DATA_BLOCK "DB92_OP_Data"
{ S7_Optimized_Access := 'FALSE' }
VERSION : 0.1
NON_RETAIN
   STRUCT
      LocTime {InstructionName := 'DTL'; LibVersion := '1.0'} : DTL;
      tm_Array : Array[0..11] of Byte;
      Msg_B0 : Array[0..63] of Word;
      CtrlJob : Array[0..3] of Word;   // Steuerungsauftragsfach
      PicNum : Array[0..4] of Word;   // Steuerungsauftragsfach
      SPS_Idx : Int;   // Index eigene SPS
      Antr_Idx : Int;   // Index ausgewählter Antrieb für Anzeige/Bedienung
      Antr_Typ : Int;   // Typ ausgewählter Antrieb für Anzeige/Bedienung
      UserPrio : Int;   // Prio 0 - keine Bedienung, Prio 1 - Antrieb einzel, Prio 2 - alle Antriebe auf Bed. UV, Prio 3 - Parametrierung
      Antr_loc_prev : Bool;   // vorhergehenden (lokal) Antrieb in Panel-Auswahl anzeigen
      Antr_loc_next : Bool;   // nächsten Antrieb (lokal) in Panel-Auswahl anzeigen
      Antr_rem_prev : Bool;   // vorhergehenden (fern) Antrieb in Panel-Auswahl anzeigen
      Antr_rem_next : Bool;   // nächsten Antrieb (fern) in Panel-Auswahl anzeigen
      UserChg : Bool;   // Panelbenutzer hat gewechselt -> remote login prüfen
      PicSet_Antr_Menu : Bool;   // UV spezifisches Menü Antriebe aufrufen
      PicSet_Antr_Prm : Bool;   // Parameterbild zum gewählten Antrieb aufrufen
      MsgQuit : Bool;   // Quittierung Meldesystem
      Antr_Text_Idx_vis : Int;   // Textlisten für Bezeichnungen - Index für Auswahl Subliste 0..3
      Antr_Text_Idx_W0 : DWord;   // Textlisten für Bezeichnungen - Subliste 0
      Antr_Text_Idx_W1 : DWord;   // Textlisten für Bezeichnungen - Subliste 1
      Antr_Text_Idx_W2 : DWord;   // Textlisten für Bezeichnungen - Subliste 2
      Antr_Text_Idx_W3 : DWord;   // Textlisten für Bezeichnungen - Subliste 3
      UserID_BitIdx : DWord;   // Benutzerkennung bitweise, ID1=Bit 1 usw.
      Antr_UV_Idx : Byte;   // Index UV des gewählten Antriebs -> Anzeige, wenn nicht in eigener SPS abgearbeitet
      SPS_Idx_BitIdx : Byte;   // Index eigene SPS - Bitliste
      Antr_UV_rem : Bool;   // Hinweisfeld, wenn Antrieb in remoter SPS bearbeitet wird
      Antr_Bed_Sperr_0 : Array[0..63] of Bool;
      Antr_Bed_Sperr_1 : Array[0..63] of Bool;
      Bed_NHV : Array[1..128] of Bool;   // Bedienberechtigungen für (ferne) OP Bedienung
      activeUserGroup : Int;
   END_STRUCT;


BEGIN

END_DATA_BLOCK

DATA_BLOCK "DB93_AntrIdx"
{ S7_Optimized_Access := 'FALSE' }
VERSION : 0.1
NON_RETAIN
   STRUCT
      MaxIdx_ges : Int;
      MaxIdx : Array[0..6] of Byte;
      UV2ZEN : Array[0..6, 1..32] of Byte;
      ZEN2UV : Array[0..6, 1..132] of Byte;
      ANTR2UV : Array[1..132] of Byte;
      ANTR2OP : Array[1..132] of Byte;
      ANTR2TYP : Array[1..132] of Byte;
   END_STRUCT;


BEGIN
   MaxIdx_ges := 22;
   MaxIdx[0] := 16#00;
   MaxIdx[1] := 16#00;
   MaxIdx[2] := 16#16;
   MaxIdx[3] := 16#00;
   MaxIdx[4] := 16#00;
   MaxIdx[5] := 16#00;
   MaxIdx[6] := 16#00;
   UV2ZEN[0,1] := 16#00;
   UV2ZEN[0,2] := 16#00;
   UV2ZEN[0,3] := 16#00;
   UV2ZEN[0,4] := 16#00;
   UV2ZEN[0,5] := 16#00;
   UV2ZEN[0,6] := 16#00;
   UV2ZEN[0,7] := 16#00;
   UV2ZEN[0,8] := 16#00;
   UV2ZEN[0,9] := 16#00;
   UV2ZEN[0,10] := 16#00;
   UV2ZEN[0,11] := 16#00;
   UV2ZEN[0,12] := 16#00;
   UV2ZEN[0,13] := 16#00;
   UV2ZEN[0,14] := 16#00;
   UV2ZEN[0,15] := 16#00;
   UV2ZEN[0,16] := 16#00;
   UV2ZEN[0,17] := 16#00;
   UV2ZEN[0,18] := 16#00;
   UV2ZEN[0,19] := 16#00;
   UV2ZEN[0,20] := 16#00;
   UV2ZEN[0,21] := 16#00;
   UV2ZEN[0,22] := 16#00;
   UV2ZEN[0,23] := 16#00;
   UV2ZEN[0,24] := 16#00;
   UV2ZEN[0,25] := 16#00;
   UV2ZEN[0,26] := 16#00;
   UV2ZEN[0,27] := 16#00;
   UV2ZEN[0,28] := 16#00;
   UV2ZEN[0,29] := 16#00;
   UV2ZEN[0,30] := 16#00;
   UV2ZEN[0,31] := 16#00;
   UV2ZEN[0,32] := 16#00;
   UV2ZEN[1,1] := 16#00;
   UV2ZEN[1,2] := 16#00;
   UV2ZEN[1,3] := 16#00;
   UV2ZEN[1,4] := 16#00;
   UV2ZEN[1,5] := 16#00;
   UV2ZEN[1,6] := 16#00;
   UV2ZEN[1,7] := 16#00;
   UV2ZEN[1,8] := 16#00;
   UV2ZEN[1,9] := 16#00;
   UV2ZEN[1,10] := 16#00;
   UV2ZEN[1,11] := 16#00;
   UV2ZEN[1,12] := 16#00;
   UV2ZEN[1,13] := 16#00;
   UV2ZEN[1,14] := 16#00;
   UV2ZEN[1,15] := 16#00;
   UV2ZEN[1,16] := 16#00;
   UV2ZEN[1,17] := 16#00;
   UV2ZEN[1,18] := 16#00;
   UV2ZEN[1,19] := 16#00;
   UV2ZEN[1,20] := 16#00;
   UV2ZEN[1,21] := 16#00;
   UV2ZEN[1,22] := 16#00;
   UV2ZEN[1,23] := 16#00;
   UV2ZEN[1,24] := 16#00;
   UV2ZEN[1,25] := 16#00;
   UV2ZEN[1,26] := 16#00;
   UV2ZEN[1,27] := 16#00;
   UV2ZEN[1,28] := 16#00;
   UV2ZEN[1,29] := 16#00;
   UV2ZEN[1,30] := 16#00;
   UV2ZEN[1,31] := 16#00;
   UV2ZEN[1,32] := 16#00;
   UV2ZEN[2,1] := 16#01;
   UV2ZEN[2,2] := 16#02;
   UV2ZEN[2,3] := 16#03;
   UV2ZEN[2,4] := 16#04;
   UV2ZEN[2,5] := 16#05;
   UV2ZEN[2,6] := 16#06;
   UV2ZEN[2,7] := 16#07;
   UV2ZEN[2,8] := 16#08;
   UV2ZEN[2,9] := 16#09;
   UV2ZEN[2,10] := 16#0A;
   UV2ZEN[2,11] := 16#0B;
   UV2ZEN[2,12] := 16#0C;
   UV2ZEN[2,13] := 16#0D;
   UV2ZEN[2,14] := 16#0E;
   UV2ZEN[2,15] := 16#0F;
   UV2ZEN[2,16] := 16#10;
   UV2ZEN[2,17] := 16#11;
   UV2ZEN[2,18] := 16#12;
   UV2ZEN[2,19] := 16#13;
   UV2ZEN[2,20] := 16#14;
   UV2ZEN[2,21] := 16#15;
   UV2ZEN[2,22] := 16#16;
   UV2ZEN[2,23] := 16#00;
   UV2ZEN[2,24] := 16#00;
   UV2ZEN[2,25] := 16#00;
   UV2ZEN[2,26] := 16#00;
   UV2ZEN[2,27] := 16#00;
   UV2ZEN[2,28] := 16#00;
   UV2ZEN[2,29] := 16#00;
   UV2ZEN[2,30] := 16#00;
   UV2ZEN[2,31] := 16#00;
   UV2ZEN[2,32] := 16#00;
   UV2ZEN[3,1] := 16#00;
   UV2ZEN[3,2] := 16#00;
   UV2ZEN[3,3] := 16#00;
   UV2ZEN[3,4] := 16#00;
   UV2ZEN[3,5] := 16#00;
   UV2ZEN[3,6] := 16#00;
   UV2ZEN[3,7] := 16#00;
   UV2ZEN[3,8] := 16#00;
   UV2ZEN[3,9] := 16#00;
   UV2ZEN[3,10] := 16#00;
   UV2ZEN[3,11] := 16#00;
   UV2ZEN[3,12] := 16#00;
   UV2ZEN[3,13] := 16#00;
   UV2ZEN[3,14] := 16#00;
   UV2ZEN[3,15] := 16#00;
   UV2ZEN[3,16] := 16#00;
   UV2ZEN[3,17] := 16#00;
   UV2ZEN[3,18] := 16#00;
   UV2ZEN[3,19] := 16#00;
   UV2ZEN[3,20] := 16#00;
   UV2ZEN[3,21] := 16#00;
   UV2ZEN[3,22] := 16#00;
   UV2ZEN[3,23] := 16#00;
   UV2ZEN[3,24] := 16#00;
   UV2ZEN[3,25] := 16#00;
   UV2ZEN[3,26] := 16#00;
   UV2ZEN[3,27] := 16#00;
   UV2ZEN[3,28] := 16#00;
   UV2ZEN[3,29] := 16#00;
   UV2ZEN[3,30] := 16#00;
   UV2ZEN[3,31] := 16#00;
   UV2ZEN[3,32] := 16#00;
   UV2ZEN[4,1] := 16#00;
   UV2ZEN[4,2] := 16#00;
   UV2ZEN[4,3] := 16#00;
   UV2ZEN[4,4] := 16#00;
   UV2ZEN[4,5] := 16#00;
   UV2ZEN[4,6] := 16#00;
   UV2ZEN[4,7] := 16#00;
   UV2ZEN[4,8] := 16#00;
   UV2ZEN[4,9] := 16#00;
   UV2ZEN[4,10] := 16#00;
   UV2ZEN[4,11] := 16#00;
   UV2ZEN[4,12] := 16#00;
   UV2ZEN[4,13] := 16#00;
   UV2ZEN[4,14] := 16#00;
   UV2ZEN[4,15] := 16#00;
   UV2ZEN[4,16] := 16#00;
   UV2ZEN[4,17] := 16#00;
   UV2ZEN[4,18] := 16#00;
   UV2ZEN[4,19] := 16#00;
   UV2ZEN[4,20] := 16#00;
   UV2ZEN[4,21] := 16#00;
   UV2ZEN[4,22] := 16#00;
   UV2ZEN[4,23] := 16#00;
   UV2ZEN[4,24] := 16#00;
   UV2ZEN[4,25] := 16#00;
   UV2ZEN[4,26] := 16#00;
   UV2ZEN[4,27] := 16#00;
   UV2ZEN[4,28] := 16#00;
   UV2ZEN[4,29] := 16#00;
   UV2ZEN[4,30] := 16#00;
   UV2ZEN[4,31] := 16#00;
   UV2ZEN[4,32] := 16#00;
   UV2ZEN[5,1] := 16#00;
   UV2ZEN[5,2] := 16#00;
   UV2ZEN[5,3] := 16#00;
   UV2ZEN[5,4] := 16#00;
   UV2ZEN[5,5] := 16#00;
   UV2ZEN[5,6] := 16#00;
   UV2ZEN[5,7] := 16#00;
   UV2ZEN[5,8] := 16#00;
   UV2ZEN[5,9] := 16#00;
   UV2ZEN[5,10] := 16#00;
   UV2ZEN[5,11] := 16#00;
   UV2ZEN[5,12] := 16#00;
   UV2ZEN[5,13] := 16#00;
   UV2ZEN[5,14] := 16#00;
   UV2ZEN[5,15] := 16#00;
   UV2ZEN[5,16] := 16#00;
   UV2ZEN[5,17] := 16#00;
   UV2ZEN[5,18] := 16#00;
   UV2ZEN[5,19] := 16#00;
   UV2ZEN[5,20] := 16#00;
   UV2ZEN[5,21] := 16#00;
   UV2ZEN[5,22] := 16#00;
   UV2ZEN[5,23] := 16#00;
   UV2ZEN[5,24] := 16#00;
   UV2ZEN[5,25] := 16#00;
   UV2ZEN[5,26] := 16#00;
   UV2ZEN[5,27] := 16#00;
   UV2ZEN[5,28] := 16#00;
   UV2ZEN[5,29] := 16#00;
   UV2ZEN[5,30] := 16#00;
   UV2ZEN[5,31] := 16#00;
   UV2ZEN[5,32] := 16#00;
   UV2ZEN[6,1] := 16#00;
   UV2ZEN[6,2] := 16#00;
   UV2ZEN[6,3] := 16#00;
   UV2ZEN[6,4] := 16#00;
   UV2ZEN[6,5] := 16#00;
   UV2ZEN[6,6] := 16#00;
   UV2ZEN[6,7] := 16#00;
   UV2ZEN[6,8] := 16#00;
   UV2ZEN[6,9] := 16#00;
   UV2ZEN[6,10] := 16#00;
   UV2ZEN[6,11] := 16#00;
   UV2ZEN[6,12] := 16#00;
   UV2ZEN[6,13] := 16#00;
   UV2ZEN[6,14] := 16#00;
   UV2ZEN[6,15] := 16#00;
   UV2ZEN[6,16] := 16#00;
   UV2ZEN[6,17] := 16#00;
   UV2ZEN[6,18] := 16#00;
   UV2ZEN[6,19] := 16#00;
   UV2ZEN[6,20] := 16#00;
   UV2ZEN[6,21] := 16#00;
   UV2ZEN[6,22] := 16#00;
   UV2ZEN[6,23] := 16#00;
   UV2ZEN[6,24] := 16#00;
   UV2ZEN[6,25] := 16#00;
   UV2ZEN[6,26] := 16#00;
   UV2ZEN[6,27] := 16#00;
   UV2ZEN[6,28] := 16#00;
   UV2ZEN[6,29] := 16#00;
   UV2ZEN[6,30] := 16#00;
   UV2ZEN[6,31] := 16#00;
   UV2ZEN[6,32] := 16#00;
   ZEN2UV[0,1] := 16#00;
   ZEN2UV[0,2] := 16#00;
   ZEN2UV[0,3] := 16#00;
   ZEN2UV[0,4] := 16#00;
   ZEN2UV[0,5] := 16#00;
   ZEN2UV[0,6] := 16#00;
   ZEN2UV[0,7] := 16#00;
   ZEN2UV[0,8] := 16#00;
   ZEN2UV[0,9] := 16#00;
   ZEN2UV[0,10] := 16#00;
   ZEN2UV[0,11] := 16#00;
   ZEN2UV[0,12] := 16#00;
   ZEN2UV[0,13] := 16#00;
   ZEN2UV[0,14] := 16#00;
   ZEN2UV[0,15] := 16#00;
   ZEN2UV[0,16] := 16#00;
   ZEN2UV[0,17] := 16#00;
   ZEN2UV[0,18] := 16#00;
   ZEN2UV[0,19] := 16#00;
   ZEN2UV[0,20] := 16#00;
   ZEN2UV[0,21] := 16#00;
   ZEN2UV[0,22] := 16#00;
   ZEN2UV[0,23] := 16#00;
   ZEN2UV[0,24] := 16#00;
   ZEN2UV[0,25] := 16#00;
   ZEN2UV[0,26] := 16#00;
   ZEN2UV[0,27] := 16#00;
   ZEN2UV[0,28] := 16#00;
   ZEN2UV[0,29] := 16#00;
   ZEN2UV[0,30] := 16#00;
   ZEN2UV[0,31] := 16#00;
   ZEN2UV[0,32] := 16#00;
   ZEN2UV[0,33] := 16#00;
   ZEN2UV[0,34] := 16#00;
   ZEN2UV[0,35] := 16#00;
   ZEN2UV[0,36] := 16#00;
   ZEN2UV[0,37] := 16#00;
   ZEN2UV[0,38] := 16#00;
   ZEN2UV[0,39] := 16#00;
   ZEN2UV[0,40] := 16#00;
   ZEN2UV[0,41] := 16#00;
   ZEN2UV[0,42] := 16#00;
   ZEN2UV[0,43] := 16#00;
   ZEN2UV[0,44] := 16#00;
   ZEN2UV[0,45] := 16#00;
   ZEN2UV[0,46] := 16#00;
   ZEN2UV[0,47] := 16#00;
   ZEN2UV[0,48] := 16#00;
   ZEN2UV[0,49] := 16#00;
   ZEN2UV[0,50] := 16#00;
   ZEN2UV[0,51] := 16#00;
   ZEN2UV[0,52] := 16#00;
   ZEN2UV[0,53] := 16#00;
   ZEN2UV[0,54] := 16#00;
   ZEN2UV[0,55] := 16#00;
   ZEN2UV[0,56] := 16#00;
   ZEN2UV[0,57] := 16#00;
   ZEN2UV[0,58] := 16#00;
   ZEN2UV[0,59] := 16#00;
   ZEN2UV[0,60] := 16#00;
   ZEN2UV[0,61] := 16#00;
   ZEN2UV[0,62] := 16#00;
   ZEN2UV[0,63] := 16#00;
   ZEN2UV[0,64] := 16#00;
   ZEN2UV[0,65] := 16#00;
   ZEN2UV[0,66] := 16#00;
   ZEN2UV[0,67] := 16#00;
   ZEN2UV[0,68] := 16#00;
   ZEN2UV[0,69] := 16#00;
   ZEN2UV[0,70] := 16#00;
   ZEN2UV[0,71] := 16#00;
   ZEN2UV[0,72] := 16#00;
   ZEN2UV[0,73] := 16#00;
   ZEN2UV[0,74] := 16#00;
   ZEN2UV[0,75] := 16#00;
   ZEN2UV[0,76] := 16#00;
   ZEN2UV[0,77] := 16#00;
   ZEN2UV[0,78] := 16#00;
   ZEN2UV[0,79] := 16#00;
   ZEN2UV[0,80] := 16#00;
   ZEN2UV[0,81] := 16#00;
   ZEN2UV[0,82] := 16#00;
   ZEN2UV[0,83] := 16#00;
   ZEN2UV[0,84] := 16#00;
   ZEN2UV[0,85] := 16#00;
   ZEN2UV[0,86] := 16#00;
   ZEN2UV[0,87] := 16#00;
   ZEN2UV[0,88] := 16#00;
   ZEN2UV[0,89] := 16#00;
   ZEN2UV[0,90] := 16#00;
   ZEN2UV[0,91] := 16#00;
   ZEN2UV[0,92] := 16#00;
   ZEN2UV[0,93] := 16#00;
   ZEN2UV[0,94] := 16#00;
   ZEN2UV[0,95] := 16#00;
   ZEN2UV[0,96] := 16#00;
   ZEN2UV[0,97] := 16#00;
   ZEN2UV[0,98] := 16#00;
   ZEN2UV[0,99] := 16#00;
   ZEN2UV[0,100] := 16#00;
   ZEN2UV[0,101] := 16#00;
   ZEN2UV[0,102] := 16#00;
   ZEN2UV[0,103] := 16#00;
   ZEN2UV[0,104] := 16#00;
   ZEN2UV[0,105] := 16#00;
   ZEN2UV[0,106] := 16#00;
   ZEN2UV[0,107] := 16#00;
   ZEN2UV[0,108] := 16#00;
   ZEN2UV[0,109] := 16#00;
   ZEN2UV[0,110] := 16#00;
   ZEN2UV[0,111] := 16#00;
   ZEN2UV[0,112] := 16#00;
   ZEN2UV[0,113] := 16#00;
   ZEN2UV[0,114] := 16#00;
   ZEN2UV[0,115] := 16#00;
   ZEN2UV[0,116] := 16#00;
   ZEN2UV[0,117] := 16#00;
   ZEN2UV[0,118] := 16#00;
   ZEN2UV[0,119] := 16#00;
   ZEN2UV[0,120] := 16#00;
   ZEN2UV[0,121] := 16#00;
   ZEN2UV[0,122] := 16#00;
   ZEN2UV[0,123] := 16#00;
   ZEN2UV[0,124] := 16#00;
   ZEN2UV[0,125] := 16#00;
   ZEN2UV[0,126] := 16#00;
   ZEN2UV[0,127] := 16#00;
   ZEN2UV[0,128] := 16#00;
   ZEN2UV[0,129] := 16#00;
   ZEN2UV[0,130] := 16#00;
   ZEN2UV[0,131] := 16#00;
   ZEN2UV[0,132] := 16#00;
   ZEN2UV[1,1] := 16#00;
   ZEN2UV[1,2] := 16#00;
   ZEN2UV[1,3] := 16#00;
   ZEN2UV[1,4] := 16#00;
   ZEN2UV[1,5] := 16#00;
   ZEN2UV[1,6] := 16#00;
   ZEN2UV[1,7] := 16#00;
   ZEN2UV[1,8] := 16#00;
   ZEN2UV[1,9] := 16#00;
   ZEN2UV[1,10] := 16#00;
   ZEN2UV[1,11] := 16#00;
   ZEN2UV[1,12] := 16#00;
   ZEN2UV[1,13] := 16#00;
   ZEN2UV[1,14] := 16#00;
   ZEN2UV[1,15] := 16#00;
   ZEN2UV[1,16] := 16#00;
   ZEN2UV[1,17] := 16#00;
   ZEN2UV[1,18] := 16#00;
   ZEN2UV[1,19] := 16#00;
   ZEN2UV[1,20] := 16#00;
   ZEN2UV[1,21] := 16#00;
   ZEN2UV[1,22] := 16#00;
   ZEN2UV[1,23] := 16#00;
   ZEN2UV[1,24] := 16#00;
   ZEN2UV[1,25] := 16#00;
   ZEN2UV[1,26] := 16#00;
   ZEN2UV[1,27] := 16#00;
   ZEN2UV[1,28] := 16#00;
   ZEN2UV[1,29] := 16#00;
   ZEN2UV[1,30] := 16#00;
   ZEN2UV[1,31] := 16#00;
   ZEN2UV[1,32] := 16#00;
   ZEN2UV[1,33] := 16#00;
   ZEN2UV[1,34] := 16#00;
   ZEN2UV[1,35] := 16#00;
   ZEN2UV[1,36] := 16#00;
   ZEN2UV[1,37] := 16#00;
   ZEN2UV[1,38] := 16#00;
   ZEN2UV[1,39] := 16#00;
   ZEN2UV[1,40] := 16#00;
   ZEN2UV[1,41] := 16#00;
   ZEN2UV[1,42] := 16#00;
   ZEN2UV[1,43] := 16#00;
   ZEN2UV[1,44] := 16#00;
   ZEN2UV[1,45] := 16#00;
   ZEN2UV[1,46] := 16#00;
   ZEN2UV[1,47] := 16#00;
   ZEN2UV[1,48] := 16#00;
   ZEN2UV[1,49] := 16#00;
   ZEN2UV[1,50] := 16#00;
   ZEN2UV[1,51] := 16#00;
   ZEN2UV[1,52] := 16#00;
   ZEN2UV[1,53] := 16#00;
   ZEN2UV[1,54] := 16#00;
   ZEN2UV[1,55] := 16#00;
   ZEN2UV[1,56] := 16#00;
   ZEN2UV[1,57] := 16#00;
   ZEN2UV[1,58] := 16#00;
   ZEN2UV[1,59] := 16#00;
   ZEN2UV[1,60] := 16#00;
   ZEN2UV[1,61] := 16#00;
   ZEN2UV[1,62] := 16#00;
   ZEN2UV[1,63] := 16#00;
   ZEN2UV[1,64] := 16#00;
   ZEN2UV[1,65] := 16#00;
   ZEN2UV[1,66] := 16#00;
   ZEN2UV[1,67] := 16#00;
   ZEN2UV[1,68] := 16#00;
   ZEN2UV[1,69] := 16#00;
   ZEN2UV[1,70] := 16#00;
   ZEN2UV[1,71] := 16#00;
   ZEN2UV[1,72] := 16#00;
   ZEN2UV[1,73] := 16#00;
   ZEN2UV[1,74] := 16#00;
   ZEN2UV[1,75] := 16#00;
   ZEN2UV[1,76] := 16#00;
   ZEN2UV[1,77] := 16#00;
   ZEN2UV[1,78] := 16#00;
   ZEN2UV[1,79] := 16#00;
   ZEN2UV[1,80] := 16#00;
   ZEN2UV[1,81] := 16#00;
   ZEN2UV[1,82] := 16#00;
   ZEN2UV[1,83] := 16#00;
   ZEN2UV[1,84] := 16#00;
   ZEN2UV[1,85] := 16#00;
   ZEN2UV[1,86] := 16#00;
   ZEN2UV[1,87] := 16#00;
   ZEN2UV[1,88] := 16#00;
   ZEN2UV[1,89] := 16#00;
   ZEN2UV[1,90] := 16#00;
   ZEN2UV[1,91] := 16#00;
   ZEN2UV[1,92] := 16#00;
   ZEN2UV[1,93] := 16#00;
   ZEN2UV[1,94] := 16#00;
   ZEN2UV[1,95] := 16#00;
   ZEN2UV[1,96] := 16#00;
   ZEN2UV[1,97] := 16#00;
   ZEN2UV[1,98] := 16#00;
   ZEN2UV[1,99] := 16#00;
   ZEN2UV[1,100] := 16#00;
   ZEN2UV[1,101] := 16#00;
   ZEN2UV[1,102] := 16#00;
   ZEN2UV[1,103] := 16#00;
   ZEN2UV[1,104] := 16#00;
   ZEN2UV[1,105] := 16#00;
   ZEN2UV[1,106] := 16#00;
   ZEN2UV[1,107] := 16#00;
   ZEN2UV[1,108] := 16#00;
   ZEN2UV[1,109] := 16#00;
   ZEN2UV[1,110] := 16#00;
   ZEN2UV[1,111] := 16#00;
   ZEN2UV[1,112] := 16#00;
   ZEN2UV[1,113] := 16#00;
   ZEN2UV[1,114] := 16#00;
   ZEN2UV[1,115] := 16#00;
   ZEN2UV[1,116] := 16#00;
   ZEN2UV[1,117] := 16#00;
   ZEN2UV[1,118] := 16#00;
   ZEN2UV[1,119] := 16#00;
   ZEN2UV[1,120] := 16#00;
   ZEN2UV[1,121] := 16#00;
   ZEN2UV[1,122] := 16#00;
   ZEN2UV[1,123] := 16#00;
   ZEN2UV[1,124] := 16#00;
   ZEN2UV[1,125] := 16#00;
   ZEN2UV[1,126] := 16#00;
   ZEN2UV[1,127] := 16#00;
   ZEN2UV[1,128] := 16#00;
   ZEN2UV[1,129] := 16#00;
   ZEN2UV[1,130] := 16#00;
   ZEN2UV[1,131] := 16#00;
   ZEN2UV[1,132] := 16#00;
   ZEN2UV[2,1] := 16#01;
   ZEN2UV[2,2] := 16#02;
   ZEN2UV[2,3] := 16#03;
   ZEN2UV[2,4] := 16#04;
   ZEN2UV[2,5] := 16#05;
   ZEN2UV[2,6] := 16#06;
   ZEN2UV[2,7] := 16#07;
   ZEN2UV[2,8] := 16#08;
   ZEN2UV[2,9] := 16#09;
   ZEN2UV[2,10] := 16#0A;
   ZEN2UV[2,11] := 16#0B;
   ZEN2UV[2,12] := 16#0C;
   ZEN2UV[2,13] := 16#0D;
   ZEN2UV[2,14] := 16#0E;
   ZEN2UV[2,15] := 16#0F;
   ZEN2UV[2,16] := 16#10;
   ZEN2UV[2,17] := 16#11;
   ZEN2UV[2,18] := 16#12;
   ZEN2UV[2,19] := 16#13;
   ZEN2UV[2,20] := 16#14;
   ZEN2UV[2,21] := 16#15;
   ZEN2UV[2,22] := 16#16;
   ZEN2UV[2,23] := 16#00;
   ZEN2UV[2,24] := 16#00;
   ZEN2UV[2,25] := 16#00;
   ZEN2UV[2,26] := 16#00;
   ZEN2UV[2,27] := 16#00;
   ZEN2UV[2,28] := 16#00;
   ZEN2UV[2,29] := 16#00;
   ZEN2UV[2,30] := 16#00;
   ZEN2UV[2,31] := 16#00;
   ZEN2UV[2,32] := 16#00;
   ZEN2UV[2,33] := 16#00;
   ZEN2UV[2,34] := 16#00;
   ZEN2UV[2,35] := 16#00;
   ZEN2UV[2,36] := 16#00;
   ZEN2UV[2,37] := 16#00;
   ZEN2UV[2,38] := 16#00;
   ZEN2UV[2,39] := 16#00;
   ZEN2UV[2,40] := 16#00;
   ZEN2UV[2,41] := 16#00;
   ZEN2UV[2,42] := 16#00;
   ZEN2UV[2,43] := 16#00;
   ZEN2UV[2,44] := 16#00;
   ZEN2UV[2,45] := 16#00;
   ZEN2UV[2,46] := 16#00;
   ZEN2UV[2,47] := 16#00;
   ZEN2UV[2,48] := 16#00;
   ZEN2UV[2,49] := 16#00;
   ZEN2UV[2,50] := 16#00;
   ZEN2UV[2,51] := 16#00;
   ZEN2UV[2,52] := 16#00;
   ZEN2UV[2,53] := 16#00;
   ZEN2UV[2,54] := 16#00;
   ZEN2UV[2,55] := 16#00;
   ZEN2UV[2,56] := 16#00;
   ZEN2UV[2,57] := 16#00;
   ZEN2UV[2,58] := 16#00;
   ZEN2UV[2,59] := 16#00;
   ZEN2UV[2,60] := 16#00;
   ZEN2UV[2,61] := 16#00;
   ZEN2UV[2,62] := 16#00;
   ZEN2UV[2,63] := 16#00;
   ZEN2UV[2,64] := 16#00;
   ZEN2UV[2,65] := 16#00;
   ZEN2UV[2,66] := 16#00;
   ZEN2UV[2,67] := 16#00;
   ZEN2UV[2,68] := 16#00;
   ZEN2UV[2,69] := 16#00;
   ZEN2UV[2,70] := 16#00;
   ZEN2UV[2,71] := 16#00;
   ZEN2UV[2,72] := 16#00;
   ZEN2UV[2,73] := 16#00;
   ZEN2UV[2,74] := 16#00;
   ZEN2UV[2,75] := 16#00;
   ZEN2UV[2,76] := 16#00;
   ZEN2UV[2,77] := 16#00;
   ZEN2UV[2,78] := 16#00;
   ZEN2UV[2,79] := 16#00;
   ZEN2UV[2,80] := 16#00;
   ZEN2UV[2,81] := 16#00;
   ZEN2UV[2,82] := 16#00;
   ZEN2UV[2,83] := 16#00;
   ZEN2UV[2,84] := 16#00;
   ZEN2UV[2,85] := 16#00;
   ZEN2UV[2,86] := 16#00;
   ZEN2UV[2,87] := 16#00;
   ZEN2UV[2,88] := 16#00;
   ZEN2UV[2,89] := 16#00;
   ZEN2UV[2,90] := 16#00;
   ZEN2UV[2,91] := 16#00;
   ZEN2UV[2,92] := 16#00;
   ZEN2UV[2,93] := 16#00;
   ZEN2UV[2,94] := 16#00;
   ZEN2UV[2,95] := 16#00;
   ZEN2UV[2,96] := 16#00;
   ZEN2UV[2,97] := 16#00;
   ZEN2UV[2,98] := 16#00;
   ZEN2UV[2,99] := 16#00;
   ZEN2UV[2,100] := 16#00;
   ZEN2UV[2,101] := 16#00;
   ZEN2UV[2,102] := 16#00;
   ZEN2UV[2,103] := 16#00;
   ZEN2UV[2,104] := 16#00;
   ZEN2UV[2,105] := 16#00;
   ZEN2UV[2,106] := 16#00;
   ZEN2UV[2,107] := 16#00;
   ZEN2UV[2,108] := 16#00;
   ZEN2UV[2,109] := 16#00;
   ZEN2UV[2,110] := 16#00;
   ZEN2UV[2,111] := 16#00;
   ZEN2UV[2,112] := 16#00;
   ZEN2UV[2,113] := 16#00;
   ZEN2UV[2,114] := 16#00;
   ZEN2UV[2,115] := 16#00;
   ZEN2UV[2,116] := 16#00;
   ZEN2UV[2,117] := 16#00;
   ZEN2UV[2,118] := 16#00;
   ZEN2UV[2,119] := 16#00;
   ZEN2UV[2,120] := 16#00;
   ZEN2UV[2,121] := 16#00;
   ZEN2UV[2,122] := 16#00;
   ZEN2UV[2,123] := 16#00;
   ZEN2UV[2,124] := 16#00;
   ZEN2UV[2,125] := 16#00;
   ZEN2UV[2,126] := 16#00;
   ZEN2UV[2,127] := 16#00;
   ZEN2UV[2,128] := 16#00;
   ZEN2UV[2,129] := 16#00;
   ZEN2UV[2,130] := 16#00;
   ZEN2UV[2,131] := 16#00;
   ZEN2UV[2,132] := 16#00;
   ZEN2UV[3,1] := 16#00;
   ZEN2UV[3,2] := 16#00;
   ZEN2UV[3,3] := 16#00;
   ZEN2UV[3,4] := 16#00;
   ZEN2UV[3,5] := 16#00;
   ZEN2UV[3,6] := 16#00;
   ZEN2UV[3,7] := 16#00;
   ZEN2UV[3,8] := 16#00;
   ZEN2UV[3,9] := 16#00;
   ZEN2UV[3,10] := 16#00;
   ZEN2UV[3,11] := 16#00;
   ZEN2UV[3,12] := 16#00;
   ZEN2UV[3,13] := 16#00;
   ZEN2UV[3,14] := 16#00;
   ZEN2UV[3,15] := 16#00;
   ZEN2UV[3,16] := 16#00;
   ZEN2UV[3,17] := 16#00;
   ZEN2UV[3,18] := 16#00;
   ZEN2UV[3,19] := 16#00;
   ZEN2UV[3,20] := 16#00;
   ZEN2UV[3,21] := 16#00;
   ZEN2UV[3,22] := 16#00;
   ZEN2UV[3,23] := 16#00;
   ZEN2UV[3,24] := 16#00;
   ZEN2UV[3,25] := 16#00;
   ZEN2UV[3,26] := 16#00;
   ZEN2UV[3,27] := 16#00;
   ZEN2UV[3,28] := 16#00;
   ZEN2UV[3,29] := 16#00;
   ZEN2UV[3,30] := 16#00;
   ZEN2UV[3,31] := 16#00;
   ZEN2UV[3,32] := 16#00;
   ZEN2UV[3,33] := 16#00;
   ZEN2UV[3,34] := 16#00;
   ZEN2UV[3,35] := 16#00;
   ZEN2UV[3,36] := 16#00;
   ZEN2UV[3,37] := 16#00;
   ZEN2UV[3,38] := 16#00;
   ZEN2UV[3,39] := 16#00;
   ZEN2UV[3,40] := 16#00;
   ZEN2UV[3,41] := 16#00;
   ZEN2UV[3,42] := 16#00;
   ZEN2UV[3,43] := 16#00;
   ZEN2UV[3,44] := 16#00;
   ZEN2UV[3,45] := 16#00;
   ZEN2UV[3,46] := 16#00;
   ZEN2UV[3,47] := 16#00;
   ZEN2UV[3,48] := 16#00;
   ZEN2UV[3,49] := 16#00;
   ZEN2UV[3,50] := 16#00;
   ZEN2UV[3,51] := 16#00;
   ZEN2UV[3,52] := 16#00;
   ZEN2UV[3,53] := 16#00;
   ZEN2UV[3,54] := 16#00;
   ZEN2UV[3,55] := 16#00;
   ZEN2UV[3,56] := 16#00;
   ZEN2UV[3,57] := 16#00;
   ZEN2UV[3,58] := 16#00;
   ZEN2UV[3,59] := 16#00;
   ZEN2UV[3,60] := 16#00;
   ZEN2UV[3,61] := 16#00;
   ZEN2UV[3,62] := 16#00;
   ZEN2UV[3,63] := 16#00;
   ZEN2UV[3,64] := 16#00;
   ZEN2UV[3,65] := 16#00;
   ZEN2UV[3,66] := 16#00;
   ZEN2UV[3,67] := 16#00;
   ZEN2UV[3,68] := 16#00;
   ZEN2UV[3,69] := 16#00;
   ZEN2UV[3,70] := 16#00;
   ZEN2UV[3,71] := 16#00;
   ZEN2UV[3,72] := 16#00;
   ZEN2UV[3,73] := 16#00;
   ZEN2UV[3,74] := 16#00;
   ZEN2UV[3,75] := 16#00;
   ZEN2UV[3,76] := 16#00;
   ZEN2UV[3,77] := 16#00;
   ZEN2UV[3,78] := 16#00;
   ZEN2UV[3,79] := 16#00;
   ZEN2UV[3,80] := 16#00;
   ZEN2UV[3,81] := 16#00;
   ZEN2UV[3,82] := 16#00;
   ZEN2UV[3,83] := 16#00;
   ZEN2UV[3,84] := 16#00;
   ZEN2UV[3,85] := 16#00;
   ZEN2UV[3,86] := 16#00;
   ZEN2UV[3,87] := 16#00;
   ZEN2UV[3,88] := 16#00;
   ZEN2UV[3,89] := 16#00;
   ZEN2UV[3,90] := 16#00;
   ZEN2UV[3,91] := 16#00;
   ZEN2UV[3,92] := 16#00;
   ZEN2UV[3,93] := 16#00;
   ZEN2UV[3,94] := 16#00;
   ZEN2UV[3,95] := 16#00;
   ZEN2UV[3,96] := 16#00;
   ZEN2UV[3,97] := 16#00;
   ZEN2UV[3,98] := 16#00;
   ZEN2UV[3,99] := 16#00;
   ZEN2UV[3,100] := 16#00;
   ZEN2UV[3,101] := 16#00;
   ZEN2UV[3,102] := 16#00;
   ZEN2UV[3,103] := 16#00;
   ZEN2UV[3,104] := 16#00;
   ZEN2UV[3,105] := 16#00;
   ZEN2UV[3,106] := 16#00;
   ZEN2UV[3,107] := 16#00;
   ZEN2UV[3,108] := 16#00;
   ZEN2UV[3,109] := 16#00;
   ZEN2UV[3,110] := 16#00;
   ZEN2UV[3,111] := 16#00;
   ZEN2UV[3,112] := 16#00;
   ZEN2UV[3,113] := 16#00;
   ZEN2UV[3,114] := 16#00;
   ZEN2UV[3,115] := 16#00;
   ZEN2UV[3,116] := 16#00;
   ZEN2UV[3,117] := 16#00;
   ZEN2UV[3,118] := 16#00;
   ZEN2UV[3,119] := 16#00;
   ZEN2UV[3,120] := 16#00;
   ZEN2UV[3,121] := 16#00;
   ZEN2UV[3,122] := 16#00;
   ZEN2UV[3,123] := 16#00;
   ZEN2UV[3,124] := 16#00;
   ZEN2UV[3,125] := 16#00;
   ZEN2UV[3,126] := 16#00;
   ZEN2UV[3,127] := 16#00;
   ZEN2UV[3,128] := 16#00;
   ZEN2UV[3,129] := 16#00;
   ZEN2UV[3,130] := 16#00;
   ZEN2UV[3,131] := 16#00;
   ZEN2UV[3,132] := 16#00;
   ZEN2UV[4,1] := 16#00;
   ZEN2UV[4,2] := 16#00;
   ZEN2UV[4,3] := 16#00;
   ZEN2UV[4,4] := 16#00;
   ZEN2UV[4,5] := 16#00;
   ZEN2UV[4,6] := 16#00;
   ZEN2UV[4,7] := 16#00;
   ZEN2UV[4,8] := 16#00;
   ZEN2UV[4,9] := 16#00;
   ZEN2UV[4,10] := 16#00;
   ZEN2UV[4,11] := 16#00;
   ZEN2UV[4,12] := 16#00;
   ZEN2UV[4,13] := 16#00;
   ZEN2UV[4,14] := 16#00;
   ZEN2UV[4,15] := 16#00;
   ZEN2UV[4,16] := 16#00;
   ZEN2UV[4,17] := 16#00;
   ZEN2UV[4,18] := 16#00;
   ZEN2UV[4,19] := 16#00;
   ZEN2UV[4,20] := 16#00;
   ZEN2UV[4,21] := 16#00;
   ZEN2UV[4,22] := 16#00;
   ZEN2UV[4,23] := 16#00;
   ZEN2UV[4,24] := 16#00;
   ZEN2UV[4,25] := 16#00;
   ZEN2UV[4,26] := 16#00;
   ZEN2UV[4,27] := 16#00;
   ZEN2UV[4,28] := 16#00;
   ZEN2UV[4,29] := 16#00;
   ZEN2UV[4,30] := 16#00;
   ZEN2UV[4,31] := 16#00;
   ZEN2UV[4,32] := 16#00;
   ZEN2UV[4,33] := 16#00;
   ZEN2UV[4,34] := 16#00;
   ZEN2UV[4,35] := 16#00;
   ZEN2UV[4,36] := 16#00;
   ZEN2UV[4,37] := 16#00;
   ZEN2UV[4,38] := 16#00;
   ZEN2UV[4,39] := 16#00;
   ZEN2UV[4,40] := 16#00;
   ZEN2UV[4,41] := 16#00;
   ZEN2UV[4,42] := 16#00;
   ZEN2UV[4,43] := 16#00;
   ZEN2UV[4,44] := 16#00;
   ZEN2UV[4,45] := 16#00;
   ZEN2UV[4,46] := 16#00;
   ZEN2UV[4,47] := 16#00;
   ZEN2UV[4,48] := 16#00;
   ZEN2UV[4,49] := 16#00;
   ZEN2UV[4,50] := 16#00;
   ZEN2UV[4,51] := 16#00;
   ZEN2UV[4,52] := 16#00;
   ZEN2UV[4,53] := 16#00;
   ZEN2UV[4,54] := 16#00;
   ZEN2UV[4,55] := 16#00;
   ZEN2UV[4,56] := 16#00;
   ZEN2UV[4,57] := 16#00;
   ZEN2UV[4,58] := 16#00;
   ZEN2UV[4,59] := 16#00;
   ZEN2UV[4,60] := 16#00;
   ZEN2UV[4,61] := 16#00;
   ZEN2UV[4,62] := 16#00;
   ZEN2UV[4,63] := 16#00;
   ZEN2UV[4,64] := 16#00;
   ZEN2UV[4,65] := 16#00;
   ZEN2UV[4,66] := 16#00;
   ZEN2UV[4,67] := 16#00;
   ZEN2UV[4,68] := 16#00;
   ZEN2UV[4,69] := 16#00;
   ZEN2UV[4,70] := 16#00;
   ZEN2UV[4,71] := 16#00;
   ZEN2UV[4,72] := 16#00;
   ZEN2UV[4,73] := 16#00;
   ZEN2UV[4,74] := 16#00;
   ZEN2UV[4,75] := 16#00;
   ZEN2UV[4,76] := 16#00;
   ZEN2UV[4,77] := 16#00;
   ZEN2UV[4,78] := 16#00;
   ZEN2UV[4,79] := 16#00;
   ZEN2UV[4,80] := 16#00;
   ZEN2UV[4,81] := 16#00;
   ZEN2UV[4,82] := 16#00;
   ZEN2UV[4,83] := 16#00;
   ZEN2UV[4,84] := 16#00;
   ZEN2UV[4,85] := 16#00;
   ZEN2UV[4,86] := 16#00;
   ZEN2UV[4,87] := 16#00;
   ZEN2UV[4,88] := 16#00;
   ZEN2UV[4,89] := 16#00;
   ZEN2UV[4,90] := 16#00;
   ZEN2UV[4,91] := 16#00;
   ZEN2UV[4,92] := 16#00;
   ZEN2UV[4,93] := 16#00;
   ZEN2UV[4,94] := 16#00;
   ZEN2UV[4,95] := 16#00;
   ZEN2UV[4,96] := 16#00;
   ZEN2UV[4,97] := 16#00;
   ZEN2UV[4,98] := 16#00;
   ZEN2UV[4,99] := 16#00;
   ZEN2UV[4,100] := 16#00;
   ZEN2UV[4,101] := 16#00;
   ZEN2UV[4,102] := 16#00;
   ZEN2UV[4,103] := 16#00;
   ZEN2UV[4,104] := 16#00;
   ZEN2UV[4,105] := 16#00;
   ZEN2UV[4,106] := 16#00;
   ZEN2UV[4,107] := 16#00;
   ZEN2UV[4,108] := 16#00;
   ZEN2UV[4,109] := 16#00;
   ZEN2UV[4,110] := 16#00;
   ZEN2UV[4,111] := 16#00;
   ZEN2UV[4,112] := 16#00;
   ZEN2UV[4,113] := 16#00;
   ZEN2UV[4,114] := 16#00;
   ZEN2UV[4,115] := 16#00;
   ZEN2UV[4,116] := 16#00;
   ZEN2UV[4,117] := 16#00;
   ZEN2UV[4,118] := 16#00;
   ZEN2UV[4,119] := 16#00;
   ZEN2UV[4,120] := 16#00;
   ZEN2UV[4,121] := 16#00;
   ZEN2UV[4,122] := 16#00;
   ZEN2UV[4,123] := 16#00;
   ZEN2UV[4,124] := 16#00;
   ZEN2UV[4,125] := 16#00;
   ZEN2UV[4,126] := 16#00;
   ZEN2UV[4,127] := 16#00;
   ZEN2UV[4,128] := 16#00;
   ZEN2UV[4,129] := 16#00;
   ZEN2UV[4,130] := 16#00;
   ZEN2UV[4,131] := 16#00;
   ZEN2UV[4,132] := 16#00;
   ZEN2UV[5,1] := 16#00;
   ZEN2UV[5,2] := 16#00;
   ZEN2UV[5,3] := 16#00;
   ZEN2UV[5,4] := 16#00;
   ZEN2UV[5,5] := 16#00;
   ZEN2UV[5,6] := 16#00;
   ZEN2UV[5,7] := 16#00;
   ZEN2UV[5,8] := 16#00;
   ZEN2UV[5,9] := 16#00;
   ZEN2UV[5,10] := 16#00;
   ZEN2UV[5,11] := 16#00;
   ZEN2UV[5,12] := 16#00;
   ZEN2UV[5,13] := 16#00;
   ZEN2UV[5,14] := 16#00;
   ZEN2UV[5,15] := 16#00;
   ZEN2UV[5,16] := 16#00;
   ZEN2UV[5,17] := 16#00;
   ZEN2UV[5,18] := 16#00;
   ZEN2UV[5,19] := 16#00;
   ZEN2UV[5,20] := 16#00;
   ZEN2UV[5,21] := 16#00;
   ZEN2UV[5,22] := 16#00;
   ZEN2UV[5,23] := 16#00;
   ZEN2UV[5,24] := 16#00;
   ZEN2UV[5,25] := 16#00;
   ZEN2UV[5,26] := 16#00;
   ZEN2UV[5,27] := 16#00;
   ZEN2UV[5,28] := 16#00;
   ZEN2UV[5,29] := 16#00;
   ZEN2UV[5,30] := 16#00;
   ZEN2UV[5,31] := 16#00;
   ZEN2UV[5,32] := 16#00;
   ZEN2UV[5,33] := 16#00;
   ZEN2UV[5,34] := 16#00;
   ZEN2UV[5,35] := 16#00;
   ZEN2UV[5,36] := 16#00;
   ZEN2UV[5,37] := 16#00;
   ZEN2UV[5,38] := 16#00;
   ZEN2UV[5,39] := 16#00;
   ZEN2UV[5,40] := 16#00;
   ZEN2UV[5,41] := 16#00;
   ZEN2UV[5,42] := 16#00;
   ZEN2UV[5,43] := 16#00;
   ZEN2UV[5,44] := 16#00;
   ZEN2UV[5,45] := 16#00;
   ZEN2UV[5,46] := 16#00;
   ZEN2UV[5,47] := 16#00;
   ZEN2UV[5,48] := 16#00;
   ZEN2UV[5,49] := 16#00;
   ZEN2UV[5,50] := 16#00;
   ZEN2UV[5,51] := 16#00;
   ZEN2UV[5,52] := 16#00;
   ZEN2UV[5,53] := 16#00;
   ZEN2UV[5,54] := 16#00;
   ZEN2UV[5,55] := 16#00;
   ZEN2UV[5,56] := 16#00;
   ZEN2UV[5,57] := 16#00;
   ZEN2UV[5,58] := 16#00;
   ZEN2UV[5,59] := 16#00;
   ZEN2UV[5,60] := 16#00;
   ZEN2UV[5,61] := 16#00;
   ZEN2UV[5,62] := 16#00;
   ZEN2UV[5,63] := 16#00;
   ZEN2UV[5,64] := 16#00;
   ZEN2UV[5,65] := 16#00;
   ZEN2UV[5,66] := 16#00;
   ZEN2UV[5,67] := 16#00;
   ZEN2UV[5,68] := 16#00;
   ZEN2UV[5,69] := 16#00;
   ZEN2UV[5,70] := 16#00;
   ZEN2UV[5,71] := 16#00;
   ZEN2UV[5,72] := 16#00;
   ZEN2UV[5,73] := 16#00;
   ZEN2UV[5,74] := 16#00;
   ZEN2UV[5,75] := 16#00;
   ZEN2UV[5,76] := 16#00;
   ZEN2UV[5,77] := 16#00;
   ZEN2UV[5,78] := 16#00;
   ZEN2UV[5,79] := 16#00;
   ZEN2UV[5,80] := 16#00;
   ZEN2UV[5,81] := 16#00;
   ZEN2UV[5,82] := 16#00;
   ZEN2UV[5,83] := 16#00;
   ZEN2UV[5,84] := 16#00;
   ZEN2UV[5,85] := 16#00;
   ZEN2UV[5,86] := 16#00;
   ZEN2UV[5,87] := 16#00;
   ZEN2UV[5,88] := 16#00;
   ZEN2UV[5,89] := 16#00;
   ZEN2UV[5,90] := 16#00;
   ZEN2UV[5,91] := 16#00;
   ZEN2UV[5,92] := 16#00;
   ZEN2UV[5,93] := 16#00;
   ZEN2UV[5,94] := 16#00;
   ZEN2UV[5,95] := 16#00;
   ZEN2UV[5,96] := 16#00;
   ZEN2UV[5,97] := 16#00;
   ZEN2UV[5,98] := 16#00;
   ZEN2UV[5,99] := 16#00;
   ZEN2UV[5,100] := 16#00;
   ZEN2UV[5,101] := 16#00;
   ZEN2UV[5,102] := 16#00;
   ZEN2UV[5,103] := 16#00;
   ZEN2UV[5,104] := 16#00;
   ZEN2UV[5,105] := 16#00;
   ZEN2UV[5,106] := 16#00;
   ZEN2UV[5,107] := 16#00;
   ZEN2UV[5,108] := 16#00;
   ZEN2UV[5,109] := 16#00;
   ZEN2UV[5,110] := 16#00;
   ZEN2UV[5,111] := 16#00;
   ZEN2UV[5,112] := 16#00;
   ZEN2UV[5,113] := 16#00;
   ZEN2UV[5,114] := 16#00;
   ZEN2UV[5,115] := 16#00;
   ZEN2UV[5,116] := 16#00;
   ZEN2UV[5,117] := 16#00;
   ZEN2UV[5,118] := 16#00;
   ZEN2UV[5,119] := 16#00;
   ZEN2UV[5,120] := 16#00;
   ZEN2UV[5,121] := 16#00;
   ZEN2UV[5,122] := 16#00;
   ZEN2UV[5,123] := 16#00;
   ZEN2UV[5,124] := 16#00;
   ZEN2UV[5,125] := 16#00;
   ZEN2UV[5,126] := 16#00;
   ZEN2UV[5,127] := 16#00;
   ZEN2UV[5,128] := 16#00;
   ZEN2UV[5,129] := 16#00;
   ZEN2UV[5,130] := 16#00;
   ZEN2UV[5,131] := 16#00;
   ZEN2UV[5,132] := 16#00;
   ZEN2UV[6,1] := 16#00;
   ZEN2UV[6,2] := 16#00;
   ZEN2UV[6,3] := 16#00;
   ZEN2UV[6,4] := 16#00;
   ZEN2UV[6,5] := 16#00;
   ZEN2UV[6,6] := 16#00;
   ZEN2UV[6,7] := 16#00;
   ZEN2UV[6,8] := 16#00;
   ZEN2UV[6,9] := 16#00;
   ZEN2UV[6,10] := 16#00;
   ZEN2UV[6,11] := 16#00;
   ZEN2UV[6,12] := 16#00;
   ZEN2UV[6,13] := 16#00;
   ZEN2UV[6,14] := 16#00;
   ZEN2UV[6,15] := 16#00;
   ZEN2UV[6,16] := 16#00;
   ZEN2UV[6,17] := 16#00;
   ZEN2UV[6,18] := 16#00;
   ZEN2UV[6,19] := 16#00;
   ZEN2UV[6,20] := 16#00;
   ZEN2UV[6,21] := 16#00;
   ZEN2UV[6,22] := 16#00;
   ZEN2UV[6,23] := 16#00;
   ZEN2UV[6,24] := 16#00;
   ZEN2UV[6,25] := 16#00;
   ZEN2UV[6,26] := 16#00;
   ZEN2UV[6,27] := 16#00;
   ZEN2UV[6,28] := 16#00;
   ZEN2UV[6,29] := 16#00;
   ZEN2UV[6,30] := 16#00;
   ZEN2UV[6,31] := 16#00;
   ZEN2UV[6,32] := 16#00;
   ZEN2UV[6,33] := 16#00;
   ZEN2UV[6,34] := 16#00;
   ZEN2UV[6,35] := 16#00;
   ZEN2UV[6,36] := 16#00;
   ZEN2UV[6,37] := 16#00;
   ZEN2UV[6,38] := 16#00;
   ZEN2UV[6,39] := 16#00;
   ZEN2UV[6,40] := 16#00;
   ZEN2UV[6,41] := 16#00;
   ZEN2UV[6,42] := 16#00;
   ZEN2UV[6,43] := 16#00;
   ZEN2UV[6,44] := 16#00;
   ZEN2UV[6,45] := 16#00;
   ZEN2UV[6,46] := 16#00;
   ZEN2UV[6,47] := 16#00;
   ZEN2UV[6,48] := 16#00;
   ZEN2UV[6,49] := 16#00;
   ZEN2UV[6,50] := 16#00;
   ZEN2UV[6,51] := 16#00;
   ZEN2UV[6,52] := 16#00;
   ZEN2UV[6,53] := 16#00;
   ZEN2UV[6,54] := 16#00;
   ZEN2UV[6,55] := 16#00;
   ZEN2UV[6,56] := 16#00;
   ZEN2UV[6,57] := 16#00;
   ZEN2UV[6,58] := 16#00;
   ZEN2UV[6,59] := 16#00;
   ZEN2UV[6,60] := 16#00;
   ZEN2UV[6,61] := 16#00;
   ZEN2UV[6,62] := 16#00;
   ZEN2UV[6,63] := 16#00;
   ZEN2UV[6,64] := 16#00;
   ZEN2UV[6,65] := 16#00;
   ZEN2UV[6,66] := 16#00;
   ZEN2UV[6,67] := 16#00;
   ZEN2UV[6,68] := 16#00;
   ZEN2UV[6,69] := 16#00;
   ZEN2UV[6,70] := 16#00;
   ZEN2UV[6,71] := 16#00;
   ZEN2UV[6,72] := 16#00;
   ZEN2UV[6,73] := 16#00;
   ZEN2UV[6,74] := 16#00;
   ZEN2UV[6,75] := 16#00;
   ZEN2UV[6,76] := 16#00;
   ZEN2UV[6,77] := 16#00;
   ZEN2UV[6,78] := 16#00;
   ZEN2UV[6,79] := 16#00;
   ZEN2UV[6,80] := 16#00;
   ZEN2UV[6,81] := 16#00;
   ZEN2UV[6,82] := 16#00;
   ZEN2UV[6,83] := 16#00;
   ZEN2UV[6,84] := 16#00;
   ZEN2UV[6,85] := 16#00;
   ZEN2UV[6,86] := 16#00;
   ZEN2UV[6,87] := 16#00;
   ZEN2UV[6,88] := 16#00;
   ZEN2UV[6,89] := 16#00;
   ZEN2UV[6,90] := 16#00;
   ZEN2UV[6,91] := 16#00;
   ZEN2UV[6,92] := 16#00;
   ZEN2UV[6,93] := 16#00;
   ZEN2UV[6,94] := 16#00;
   ZEN2UV[6,95] := 16#00;
   ZEN2UV[6,96] := 16#00;
   ZEN2UV[6,97] := 16#00;
   ZEN2UV[6,98] := 16#00;
   ZEN2UV[6,99] := 16#00;
   ZEN2UV[6,100] := 16#00;
   ZEN2UV[6,101] := 16#00;
   ZEN2UV[6,102] := 16#00;
   ZEN2UV[6,103] := 16#00;
   ZEN2UV[6,104] := 16#00;
   ZEN2UV[6,105] := 16#00;
   ZEN2UV[6,106] := 16#00;
   ZEN2UV[6,107] := 16#00;
   ZEN2UV[6,108] := 16#00;
   ZEN2UV[6,109] := 16#00;
   ZEN2UV[6,110] := 16#00;
   ZEN2UV[6,111] := 16#00;
   ZEN2UV[6,112] := 16#00;
   ZEN2UV[6,113] := 16#00;
   ZEN2UV[6,114] := 16#00;
   ZEN2UV[6,115] := 16#00;
   ZEN2UV[6,116] := 16#00;
   ZEN2UV[6,117] := 16#00;
   ZEN2UV[6,118] := 16#00;
   ZEN2UV[6,119] := 16#00;
   ZEN2UV[6,120] := 16#00;
   ZEN2UV[6,121] := 16#00;
   ZEN2UV[6,122] := 16#00;
   ZEN2UV[6,123] := 16#00;
   ZEN2UV[6,124] := 16#00;
   ZEN2UV[6,125] := 16#00;
   ZEN2UV[6,126] := 16#00;
   ZEN2UV[6,127] := 16#00;
   ZEN2UV[6,128] := 16#00;
   ZEN2UV[6,129] := 16#00;
   ZEN2UV[6,130] := 16#00;
   ZEN2UV[6,131] := 16#00;
   ZEN2UV[6,132] := 16#00;
   ANTR2UV[1] := 16#02;
   ANTR2UV[2] := 16#02;
   ANTR2UV[3] := 16#02;
   ANTR2UV[4] := 16#02;
   ANTR2UV[5] := 16#02;
   ANTR2UV[6] := 16#02;
   ANTR2UV[7] := 16#02;
   ANTR2UV[8] := 16#02;
   ANTR2UV[9] := 16#02;
   ANTR2UV[10] := 16#02;
   ANTR2UV[11] := 16#02;
   ANTR2UV[12] := 16#02;
   ANTR2UV[13] := 16#02;
   ANTR2UV[14] := 16#02;
   ANTR2UV[15] := 16#02;
   ANTR2UV[16] := 16#02;
   ANTR2UV[17] := 16#02;
   ANTR2UV[18] := 16#02;
   ANTR2UV[19] := 16#02;
   ANTR2UV[20] := 16#02;
   ANTR2UV[21] := 16#02;
   ANTR2UV[22] := 16#02;
   ANTR2UV[23] := 16#00;
   ANTR2UV[24] := 16#00;
   ANTR2UV[25] := 16#00;
   ANTR2UV[26] := 16#00;
   ANTR2UV[27] := 16#00;
   ANTR2UV[28] := 16#00;
   ANTR2UV[29] := 16#00;
   ANTR2UV[30] := 16#00;
   ANTR2UV[31] := 16#00;
   ANTR2UV[32] := 16#00;
   ANTR2UV[33] := 16#00;
   ANTR2UV[34] := 16#00;
   ANTR2UV[35] := 16#00;
   ANTR2UV[36] := 16#00;
   ANTR2UV[37] := 16#00;
   ANTR2UV[38] := 16#00;
   ANTR2UV[39] := 16#00;
   ANTR2UV[40] := 16#00;
   ANTR2UV[41] := 16#00;
   ANTR2UV[42] := 16#00;
   ANTR2UV[43] := 16#00;
   ANTR2UV[44] := 16#00;
   ANTR2UV[45] := 16#00;
   ANTR2UV[46] := 16#00;
   ANTR2UV[47] := 16#00;
   ANTR2UV[48] := 16#00;
   ANTR2UV[49] := 16#00;
   ANTR2UV[50] := 16#00;
   ANTR2UV[51] := 16#00;
   ANTR2UV[52] := 16#00;
   ANTR2UV[53] := 16#00;
   ANTR2UV[54] := 16#00;
   ANTR2UV[55] := 16#00;
   ANTR2UV[56] := 16#00;
   ANTR2UV[57] := 16#00;
   ANTR2UV[58] := 16#00;
   ANTR2UV[59] := 16#00;
   ANTR2UV[60] := 16#00;
   ANTR2UV[61] := 16#00;
   ANTR2UV[62] := 16#00;
   ANTR2UV[63] := 16#00;
   ANTR2UV[64] := 16#00;
   ANTR2UV[65] := 16#00;
   ANTR2UV[66] := 16#00;
   ANTR2UV[67] := 16#00;
   ANTR2UV[68] := 16#00;
   ANTR2UV[69] := 16#00;
   ANTR2UV[70] := 16#00;
   ANTR2UV[71] := 16#00;
   ANTR2UV[72] := 16#00;
   ANTR2UV[73] := 16#00;
   ANTR2UV[74] := 16#00;
   ANTR2UV[75] := 16#00;
   ANTR2UV[76] := 16#00;
   ANTR2UV[77] := 16#00;
   ANTR2UV[78] := 16#00;
   ANTR2UV[79] := 16#00;
   ANTR2UV[80] := 16#00;
   ANTR2UV[81] := 16#00;
   ANTR2UV[82] := 16#00;
   ANTR2UV[83] := 16#00;
   ANTR2UV[84] := 16#00;
   ANTR2UV[85] := 16#00;
   ANTR2UV[86] := 16#00;
   ANTR2UV[87] := 16#00;
   ANTR2UV[88] := 16#00;
   ANTR2UV[89] := 16#00;
   ANTR2UV[90] := 16#00;
   ANTR2UV[91] := 16#00;
   ANTR2UV[92] := 16#00;
   ANTR2UV[93] := 16#00;
   ANTR2UV[94] := 16#00;
   ANTR2UV[95] := 16#00;
   ANTR2UV[96] := 16#00;
   ANTR2UV[97] := 16#00;
   ANTR2UV[98] := 16#00;
   ANTR2UV[99] := 16#00;
   ANTR2UV[100] := 16#00;
   ANTR2UV[101] := 16#00;
   ANTR2UV[102] := 16#00;
   ANTR2UV[103] := 16#00;
   ANTR2UV[104] := 16#00;
   ANTR2UV[105] := 16#00;
   ANTR2UV[106] := 16#00;
   ANTR2UV[107] := 16#00;
   ANTR2UV[108] := 16#00;
   ANTR2UV[109] := 16#00;
   ANTR2UV[110] := 16#00;
   ANTR2UV[111] := 16#00;
   ANTR2UV[112] := 16#00;
   ANTR2UV[113] := 16#00;
   ANTR2UV[114] := 16#00;
   ANTR2UV[115] := 16#00;
   ANTR2UV[116] := 16#00;
   ANTR2UV[117] := 16#00;
   ANTR2UV[118] := 16#00;
   ANTR2UV[119] := 16#00;
   ANTR2UV[120] := 16#00;
   ANTR2UV[121] := 16#00;
   ANTR2UV[122] := 16#00;
   ANTR2UV[123] := 16#00;
   ANTR2UV[124] := 16#00;
   ANTR2UV[125] := 16#00;
   ANTR2UV[126] := 16#00;
   ANTR2UV[127] := 16#00;
   ANTR2UV[128] := 16#00;
   ANTR2UV[129] := 16#00;
   ANTR2UV[130] := 16#00;
   ANTR2UV[131] := 16#00;
   ANTR2UV[132] := 16#00;
   ANTR2OP[1] := 16#01;
   ANTR2OP[2] := 16#01;
   ANTR2OP[3] := 16#01;
   ANTR2OP[4] := 16#01;
   ANTR2OP[5] := 16#01;
   ANTR2OP[6] := 16#01;
   ANTR2OP[7] := 16#01;
   ANTR2OP[8] := 16#01;
   ANTR2OP[9] := 16#01;
   ANTR2OP[10] := 16#01;
   ANTR2OP[11] := 16#01;
   ANTR2OP[12] := 16#01;
   ANTR2OP[13] := 16#01;
   ANTR2OP[14] := 16#01;
   ANTR2OP[15] := 16#01;
   ANTR2OP[16] := 16#01;
   ANTR2OP[17] := 16#01;
   ANTR2OP[18] := 16#01;
   ANTR2OP[19] := 16#01;
   ANTR2OP[20] := 16#01;
   ANTR2OP[21] := 16#01;
   ANTR2OP[22] := 16#01;
   ANTR2OP[23] := 16#00;
   ANTR2OP[24] := 16#00;
   ANTR2OP[25] := 16#00;
   ANTR2OP[26] := 16#00;
   ANTR2OP[27] := 16#00;
   ANTR2OP[28] := 16#00;
   ANTR2OP[29] := 16#00;
   ANTR2OP[30] := 16#00;
   ANTR2OP[31] := 16#00;
   ANTR2OP[32] := 16#00;
   ANTR2OP[33] := 16#00;
   ANTR2OP[34] := 16#00;
   ANTR2OP[35] := 16#00;
   ANTR2OP[36] := 16#00;
   ANTR2OP[37] := 16#00;
   ANTR2OP[38] := 16#00;
   ANTR2OP[39] := 16#00;
   ANTR2OP[40] := 16#00;
   ANTR2OP[41] := 16#00;
   ANTR2OP[42] := 16#00;
   ANTR2OP[43] := 16#00;
   ANTR2OP[44] := 16#00;
   ANTR2OP[45] := 16#00;
   ANTR2OP[46] := 16#00;
   ANTR2OP[47] := 16#00;
   ANTR2OP[48] := 16#00;
   ANTR2OP[49] := 16#00;
   ANTR2OP[50] := 16#00;
   ANTR2OP[51] := 16#00;
   ANTR2OP[52] := 16#00;
   ANTR2OP[53] := 16#00;
   ANTR2OP[54] := 16#00;
   ANTR2OP[55] := 16#00;
   ANTR2OP[56] := 16#00;
   ANTR2OP[57] := 16#00;
   ANTR2OP[58] := 16#00;
   ANTR2OP[59] := 16#00;
   ANTR2OP[60] := 16#00;
   ANTR2OP[61] := 16#00;
   ANTR2OP[62] := 16#00;
   ANTR2OP[63] := 16#00;
   ANTR2OP[64] := 16#00;
   ANTR2OP[65] := 16#00;
   ANTR2OP[66] := 16#00;
   ANTR2OP[67] := 16#00;
   ANTR2OP[68] := 16#00;
   ANTR2OP[69] := 16#00;
   ANTR2OP[70] := 16#00;
   ANTR2OP[71] := 16#00;
   ANTR2OP[72] := 16#00;
   ANTR2OP[73] := 16#00;
   ANTR2OP[74] := 16#00;
   ANTR2OP[75] := 16#00;
   ANTR2OP[76] := 16#00;
   ANTR2OP[77] := 16#00;
   ANTR2OP[78] := 16#00;
   ANTR2OP[79] := 16#00;
   ANTR2OP[80] := 16#00;
   ANTR2OP[81] := 16#00;
   ANTR2OP[82] := 16#00;
   ANTR2OP[83] := 16#00;
   ANTR2OP[84] := 16#00;
   ANTR2OP[85] := 16#00;
   ANTR2OP[86] := 16#00;
   ANTR2OP[87] := 16#00;
   ANTR2OP[88] := 16#00;
   ANTR2OP[89] := 16#00;
   ANTR2OP[90] := 16#00;
   ANTR2OP[91] := 16#00;
   ANTR2OP[92] := 16#00;
   ANTR2OP[93] := 16#00;
   ANTR2OP[94] := 16#00;
   ANTR2OP[95] := 16#00;
   ANTR2OP[96] := 16#00;
   ANTR2OP[97] := 16#00;
   ANTR2OP[98] := 16#00;
   ANTR2OP[99] := 16#00;
   ANTR2OP[100] := 16#00;
   ANTR2OP[101] := 16#00;
   ANTR2OP[102] := 16#00;
   ANTR2OP[103] := 16#00;
   ANTR2OP[104] := 16#00;
   ANTR2OP[105] := 16#00;
   ANTR2OP[106] := 16#00;
   ANTR2OP[107] := 16#00;
   ANTR2OP[108] := 16#00;
   ANTR2OP[109] := 16#00;
   ANTR2OP[110] := 16#00;
   ANTR2OP[111] := 16#00;
   ANTR2OP[112] := 16#00;
   ANTR2OP[113] := 16#00;
   ANTR2OP[114] := 16#00;
   ANTR2OP[115] := 16#00;
   ANTR2OP[116] := 16#00;
   ANTR2OP[117] := 16#00;
   ANTR2OP[118] := 16#00;
   ANTR2OP[119] := 16#00;
   ANTR2OP[120] := 16#00;
   ANTR2OP[121] := 16#00;
   ANTR2OP[122] := 16#00;
   ANTR2OP[123] := 16#00;
   ANTR2OP[124] := 16#00;
   ANTR2OP[125] := 16#00;
   ANTR2OP[126] := 16#00;
   ANTR2OP[127] := 16#00;
   ANTR2OP[128] := 16#00;
   ANTR2OP[129] := 16#00;
   ANTR2OP[130] := 16#00;
   ANTR2OP[131] := 16#00;
   ANTR2OP[132] := 16#00;
   ANTR2TYP[1] := 16#06;
   ANTR2TYP[2] := 16#06;
   ANTR2TYP[3] := 16#06;
   ANTR2TYP[4] := 16#06;
   ANTR2TYP[5] := 16#00;
   ANTR2TYP[6] := 16#00;
   ANTR2TYP[7] := 16#05;
   ANTR2TYP[8] := 16#05;
   ANTR2TYP[9] := 16#05;
   ANTR2TYP[10] := 16#05;
   ANTR2TYP[11] := 16#05;
   ANTR2TYP[12] := 16#05;
   ANTR2TYP[13] := 16#05;
   ANTR2TYP[14] := 16#05;
   ANTR2TYP[15] := 16#05;
   ANTR2TYP[16] := 16#05;
   ANTR2TYP[17] := 16#05;
   ANTR2TYP[18] := 16#05;
   ANTR2TYP[19] := 16#07;
   ANTR2TYP[20] := 16#07;
   ANTR2TYP[21] := 16#00;
   ANTR2TYP[22] := 16#00;
   ANTR2TYP[23] := 16#00;
   ANTR2TYP[24] := 16#00;
   ANTR2TYP[25] := 16#00;
   ANTR2TYP[26] := 16#00;
   ANTR2TYP[27] := 16#00;
   ANTR2TYP[28] := 16#00;
   ANTR2TYP[29] := 16#00;
   ANTR2TYP[30] := 16#00;
   ANTR2TYP[31] := 16#00;
   ANTR2TYP[32] := 16#00;
   ANTR2TYP[33] := 16#00;
   ANTR2TYP[34] := 16#00;
   ANTR2TYP[35] := 16#00;
   ANTR2TYP[36] := 16#00;
   ANTR2TYP[37] := 16#00;
   ANTR2TYP[38] := 16#00;
   ANTR2TYP[39] := 16#00;
   ANTR2TYP[40] := 16#00;
   ANTR2TYP[41] := 16#00;
   ANTR2TYP[42] := 16#00;
   ANTR2TYP[43] := 16#00;
   ANTR2TYP[44] := 16#00;
   ANTR2TYP[45] := 16#00;
   ANTR2TYP[46] := 16#00;
   ANTR2TYP[47] := 16#00;
   ANTR2TYP[48] := 16#00;
   ANTR2TYP[49] := 16#00;
   ANTR2TYP[50] := 16#00;
   ANTR2TYP[51] := 16#00;
   ANTR2TYP[52] := 16#00;
   ANTR2TYP[53] := 16#00;
   ANTR2TYP[54] := 16#00;
   ANTR2TYP[55] := 16#00;
   ANTR2TYP[56] := 16#00;
   ANTR2TYP[57] := 16#00;
   ANTR2TYP[58] := 16#00;
   ANTR2TYP[59] := 16#00;
   ANTR2TYP[60] := 16#00;
   ANTR2TYP[61] := 16#00;
   ANTR2TYP[62] := 16#00;
   ANTR2TYP[63] := 16#00;
   ANTR2TYP[64] := 16#00;
   ANTR2TYP[65] := 16#00;
   ANTR2TYP[66] := 16#00;
   ANTR2TYP[67] := 16#00;
   ANTR2TYP[68] := 16#00;
   ANTR2TYP[69] := 16#00;
   ANTR2TYP[70] := 16#00;
   ANTR2TYP[71] := 16#00;
   ANTR2TYP[72] := 16#00;
   ANTR2TYP[73] := 16#00;
   ANTR2TYP[74] := 16#00;
   ANTR2TYP[75] := 16#00;
   ANTR2TYP[76] := 16#00;
   ANTR2TYP[77] := 16#00;
   ANTR2TYP[78] := 16#00;
   ANTR2TYP[79] := 16#00;
   ANTR2TYP[80] := 16#00;
   ANTR2TYP[81] := 16#00;
   ANTR2TYP[82] := 16#00;
   ANTR2TYP[83] := 16#00;
   ANTR2TYP[84] := 16#00;
   ANTR2TYP[85] := 16#00;
   ANTR2TYP[86] := 16#00;
   ANTR2TYP[87] := 16#00;
   ANTR2TYP[88] := 16#00;
   ANTR2TYP[89] := 16#00;
   ANTR2TYP[90] := 16#00;
   ANTR2TYP[91] := 16#00;
   ANTR2TYP[92] := 16#00;
   ANTR2TYP[93] := 16#00;
   ANTR2TYP[94] := 16#00;
   ANTR2TYP[95] := 16#00;
   ANTR2TYP[96] := 16#00;
   ANTR2TYP[97] := 16#00;
   ANTR2TYP[98] := 16#00;
   ANTR2TYP[99] := 16#00;
   ANTR2TYP[100] := 16#00;
   ANTR2TYP[101] := 16#00;
   ANTR2TYP[102] := 16#00;
   ANTR2TYP[103] := 16#00;
   ANTR2TYP[104] := 16#00;
   ANTR2TYP[105] := 16#00;
   ANTR2TYP[106] := 16#00;
   ANTR2TYP[107] := 16#00;
   ANTR2TYP[108] := 16#00;
   ANTR2TYP[109] := 16#00;
   ANTR2TYP[110] := 16#00;
   ANTR2TYP[111] := 16#00;
   ANTR2TYP[112] := 16#00;
   ANTR2TYP[113] := 16#00;
   ANTR2TYP[114] := 16#00;
   ANTR2TYP[115] := 16#00;
   ANTR2TYP[116] := 16#00;
   ANTR2TYP[117] := 16#00;
   ANTR2TYP[118] := 16#00;
   ANTR2TYP[119] := 16#00;
   ANTR2TYP[120] := 16#00;
   ANTR2TYP[121] := 16#00;
   ANTR2TYP[122] := 16#00;
   ANTR2TYP[123] := 16#00;
   ANTR2TYP[124] := 16#00;
   ANTR2TYP[125] := 16#00;
   ANTR2TYP[126] := 16#00;
   ANTR2TYP[127] := 16#00;
   ANTR2TYP[128] := 16#00;
   ANTR2TYP[129] := 16#00;
   ANTR2TYP[130] := 16#00;
   ANTR2TYP[131] := 16#00;
   ANTR2TYP[132] := 16#00;

END_DATA_BLOCK

DATA_BLOCK "DB104_Antriebe_Meld"
{ S7_Optimized_Access := 'FALSE' }
VERSION : 0.1
   STRUCT
      BB_G1 : "T_ANTRIEB_MELD";   // Belebung - Gebläse 1
      BB_G2 : "T_ANTRIEB_MELD";   // Belebung - Gebläse 2
      BB_G3 : "T_ANTRIEB_MELD";   // Belebung - Gebläse 3
      BB_SHL_G1 : "T_ANTRIEB_MELD";   // Belebung - Schallhaubenlüfter Gebläse 1
      BB_SHL_G2 : "T_ANTRIEB_MELD";   // Belebung - Schallhaubenlüfter Gebläse 2
      BB_SHL_G3 : "T_ANTRIEB_MELD";   // Belebung - Schallhaubenlüfter Gebläse 3
      BB_AV : "T_ANTRIEB_MELD";   // Belebung - Gebläsestation - Abluftventilator
      BB_LS1 : "T_ANTRIEB_MELD";   // Belebung - Gebläsestation - Luftwegschieber 1
      BB_LS2 : "T_ANTRIEB_MELD";   // Belebung - Gebläsestation - Luftwegschieber 2
      BB1_RZP1 : "T_ANTRIEB_MELD";   // Becken 1 - Rezipumpe 1
      BB1_RZP2 : "T_ANTRIEB_MELD";   // Becken 1 - Rezipumpe 2
      BB1_UeSP : "T_ANTRIEB_MELD";   // Becken 1 - ÜSS-Pumpe
      BB1_AS1 : "T_ANTRIEB_MELD";   // Becken 1 - Ablaufschieber 1
      BB1_AS2 : "T_ANTRIEB_MELD";   // Becken 1 - Ablaufschieber 2
      BB1_SR1 : "T_ANTRIEB_MELD";   // Becken 1 - MV Schlammrückführung 1
      BB1_SR2 : "T_ANTRIEB_MELD";   // Becken 1 - MV Schlammrückführung 2
      BB2_RZP1 : "T_ANTRIEB_MELD";   // Becken 2 - Rezipumpe 1
      BB2_RZP2 : "T_ANTRIEB_MELD";   // Becken 2 - Rezipumpe 2
      BB2_UeSP : "T_ANTRIEB_MELD";   // Becken 2 - ÜSS-Pumpe
      BB2_AS1 : "T_ANTRIEB_MELD";   // Becken 2 - Ablaufschieber 1
      BB2_AS2 : "T_ANTRIEB_MELD";   // Becken 2 - Ablaufschieber 2
      BB2_SR1 : "T_ANTRIEB_MELD";   // Becken 2 - MV Schlammrückführung 1
      BB2_SR2 : "T_ANTRIEB_MELD";   // Becken 2 - MV Schlammrückführung 2
      BB1_SR_K : "T_ANTRIEB_MELD";   // Becken 1- Druckluftkompressor Schlammrückführung
      Zulauf_AR_P1 : "T_ANTRIEB_MELD";   // Zulauf - Pumpwerk "Alter Rechen" - Pumpe 1
      Zulauf_AR_P2 : "T_ANTRIEB_MELD";   // Zulauf - Pumpwerk "Alter Rechen" - Pumpe 2
      Zulauf_AS : "T_ANTRIEB_MELD";   // Zulauf - Vorlagebehälter - Absperrschieber
      Zulauf_RA_SA : "T_ANTRIEB_MELD";   // Zulauf - Rechen - Sieb
      Zulauf_RA_HZS : "T_ANTRIEB_MELD";   // Zulauf - Rechen - HZS
      Zulauf_RA_VKS : "T_ANTRIEB_MELD";   // Zulauf - Rechen - VZS
      Zulauf_RA_V : "T_ANTRIEB_MELD";   // Zulauf - Rechen - Belüfter
      Zulauf_RA_RP : "T_ANTRIEB_MELD";   // Zulauf - Rechen - Räumpaddel
      Zulauf_RA_FP : "T_ANTRIEB_MELD";   // Zulauf - Rechen - Fettpumpe
      Schlamm_BP : "T_ANTRIEB_MELD";   // Schlamm - Beschickungspumpe Schlammbeete
      Truebwasser_P1 : "T_ANTRIEB_MELD";   // Trübwasserpumpwerk - Pumpe 1
      Truebwasser_P2 : "T_ANTRIEB_MELD";   // Trübwasserpumpwerk - Pumpe 2
      Schlamm_AS : "T_ANTRIEB_MELD";   // Schlamm - Absperrschieber Schlammbeete
      BB2_SR_K : "T_ANTRIEB_MELD";   // Becken 2 - Druckluftkompressor Schlammrückführung
      Zulauf_DosP : "T_ANTRIEB_MELD";   // Zulauf - Dosierpumpe
   END_STRUCT;


BEGIN
   BB_G1.Status.Bed_vOrt := FALSE;
   BB_G1.Status.Bed_UV := FALSE;
   BB_G1.Status.Bed_NHV := FALSE;
   BB_G1.Status.Bed_PLS := TRUE;
   BB_G1.Status.BA_Hand := FALSE;
   BB_G1.Status.BA_Auto := TRUE;
   BB_G1.Status.RB_Ein1 := TRUE;
   BB_G1.Status.RB_Ein2 := FALSE;
   BB_G1.Status.RB_Aus := FALSE;
   BB_G1.Status.BFR_NS := FALSE;
   BB_G1.Status.BFR_ECS := FALSE;
   BB_G1.Status.BFR_ESK := FALSE;
   BB_G1.Status.BFR_MAZ := FALSE;
   BB_G1.Status.BFR_Rev := FALSE;
   BB_G1.Status.BFR_Ein1 := FALSE;
   BB_G1.Status.BFR_Ein2 := FALSE;
   BB_G1.Status.BM_Ein1 := TRUE;
   BB_G1.Status.BM_Ein2 := FALSE;
   BB_G1.Status.BM_Auf := FALSE;
   BB_G1.Status.BM_Zu := FALSE;
   BB_G1.Status.BM_Ein := TRUE;
   BB_G1.Status.BM_Aus := FALSE;
   BB_G1.Status.BM_Anst1 := TRUE;
   BB_G1.Status.BM_Anst2 := FALSE;
   BB_G1.Status.BM_Auto1 := TRUE;
   BB_G1.Status.BM_Auto2 := FALSE;
   BB_G1.Status.Res_26 := FALSE;
   BB_G1.Status.Res_27 := FALSE;
   BB_G1.Status.BB_NA := FALSE;
   BB_G1.Status.BB_AutoOk := TRUE;
   BB_G1.Status.BB_SS := FALSE;
   BB_G1.Status.BB_SSnq := FALSE;
   BB_G1.Stoerung.St_allg := FALSE;
   BB_G1.Stoerung.St_DMA := FALSE;
   BB_G1.Stoerung.St_DMZ := FALSE;
   BB_G1.Stoerung.St_FU := FALSE;
   BB_G1.Stoerung.St_TL := FALSE;
   BB_G1.Stoerung.St_UDr := FALSE;
   BB_G1.Stoerung.St_UeDr := FALSE;
   BB_G1.Stoerung.St_UeTemp := FALSE;
   BB_G1.Stoerung.St_Leck := FALSE;
   BB_G1.Stoerung.St_UeLM := FALSE;
   BB_G1.Stoerung.St_UeLE := FALSE;
   BB_G1.Stoerung.St_Kom_DP := FALSE;
   BB_G1.Stoerung.St_Kom_int := FALSE;
   BB_G1.Stoerung.St_int := FALSE;
   BB_G1.Stoerung.St_LZ := FALSE;
   BB_G1.Stoerung.St_BefLZ := FALSE;
   BB_G1.Stoerung.Wa_EZ := FALSE;
   BB_G1.Stoerung.Wa_Wart := FALSE;
   BB_G1.Stoerung.St_Strm := FALSE;
   BB_G1.Stoerung.Res_19 := FALSE;
   BB_G1.Stoerung.Res_20 := FALSE;
   BB_G1.Stoerung.Res_21 := FALSE;
   BB_G1.Stoerung.Res_22 := FALSE;
   BB_G1.Stoerung.Res_23 := FALSE;
   BB_G1.Stoerung.Res_24 := FALSE;
   BB_G1.Stoerung.Res_25 := FALSE;
   BB_G1.Stoerung.Res_26 := FALSE;
   BB_G1.Stoerung.Res_27 := FALSE;
   BB_G1.Stoerung.Res_28 := FALSE;
   BB_G1.Stoerung.Res_29 := FALSE;
   BB_G1.Stoerung.Res_30 := FALSE;
   BB_G1.Stoerung.Res_31 := FALSE;
   BB_G1.MW_I := 39.9;
   BB_G1.MW_P := 12.9;
   BB_G1.EZ := 0;
   BB_G1.BZ_akt := 985;
   BB_G1.BZ_ges := 287586;
   BB_G1.AZ_akt := 1196;
   BB_G1.ESH := 298;
   BB_G1.SW_akt := 6500.0;
   BB_G1.SW_Auto := 6500.0;
   BB_G1.SW_out := 6500.0;
   BB_G2.Status.Bed_vOrt := FALSE;
   BB_G2.Status.Bed_UV := FALSE;
   BB_G2.Status.Bed_NHV := FALSE;
   BB_G2.Status.Bed_PLS := TRUE;
   BB_G2.Status.BA_Hand := FALSE;
   BB_G2.Status.BA_Auto := TRUE;
   BB_G2.Status.RB_Ein1 := FALSE;
   BB_G2.Status.RB_Ein2 := FALSE;
   BB_G2.Status.RB_Aus := TRUE;
   BB_G2.Status.BFR_NS := FALSE;
   BB_G2.Status.BFR_ECS := FALSE;
   BB_G2.Status.BFR_ESK := FALSE;
   BB_G2.Status.BFR_MAZ := FALSE;
   BB_G2.Status.BFR_Rev := FALSE;
   BB_G2.Status.BFR_Ein1 := TRUE;
   BB_G2.Status.BFR_Ein2 := FALSE;
   BB_G2.Status.BM_Ein1 := FALSE;
   BB_G2.Status.BM_Ein2 := FALSE;
   BB_G2.Status.BM_Auf := FALSE;
   BB_G2.Status.BM_Zu := FALSE;
   BB_G2.Status.BM_Ein := FALSE;
   BB_G2.Status.BM_Aus := TRUE;
   BB_G2.Status.BM_Anst1 := FALSE;
   BB_G2.Status.BM_Anst2 := FALSE;
   BB_G2.Status.BM_Auto1 := TRUE;
   BB_G2.Status.BM_Auto2 := FALSE;
   BB_G2.Status.Res_26 := FALSE;
   BB_G2.Status.Res_27 := FALSE;
   BB_G2.Status.BB_NA := TRUE;
   BB_G2.Status.BB_AutoOk := FALSE;
   BB_G2.Status.BB_SS := FALSE;
   BB_G2.Status.BB_SSnq := FALSE;
   BB_G2.Stoerung.St_allg := FALSE;
   BB_G2.Stoerung.St_DMA := FALSE;
   BB_G2.Stoerung.St_DMZ := FALSE;
   BB_G2.Stoerung.St_FU := FALSE;
   BB_G2.Stoerung.St_TL := FALSE;
   BB_G2.Stoerung.St_UDr := FALSE;
   BB_G2.Stoerung.St_UeDr := FALSE;
   BB_G2.Stoerung.St_UeTemp := FALSE;
   BB_G2.Stoerung.St_Leck := FALSE;
   BB_G2.Stoerung.St_UeLM := FALSE;
   BB_G2.Stoerung.St_UeLE := FALSE;
   BB_G2.Stoerung.St_Kom_DP := FALSE;
   BB_G2.Stoerung.St_Kom_int := FALSE;
   BB_G2.Stoerung.St_int := FALSE;
   BB_G2.Stoerung.St_LZ := FALSE;
   BB_G2.Stoerung.St_BefLZ := FALSE;
   BB_G2.Stoerung.Wa_EZ := FALSE;
   BB_G2.Stoerung.Wa_Wart := FALSE;
   BB_G2.Stoerung.St_Strm := FALSE;
   BB_G2.Stoerung.Res_19 := FALSE;
   BB_G2.Stoerung.Res_20 := FALSE;
   BB_G2.Stoerung.Res_21 := FALSE;
   BB_G2.Stoerung.Res_22 := FALSE;
   BB_G2.Stoerung.Res_23 := FALSE;
   BB_G2.Stoerung.Res_24 := FALSE;
   BB_G2.Stoerung.Res_25 := FALSE;
   BB_G2.Stoerung.Res_26 := FALSE;
   BB_G2.Stoerung.Res_27 := FALSE;
   BB_G2.Stoerung.Res_28 := FALSE;
   BB_G2.Stoerung.Res_29 := FALSE;
   BB_G2.Stoerung.Res_30 := FALSE;
   BB_G2.Stoerung.Res_31 := FALSE;
   BB_G2.MW_I := 0.0;
   BB_G2.MW_P := 0.0;
   BB_G2.EZ := 0;
   BB_G2.BZ_akt := 0;
   BB_G2.BZ_ges := 376975;
   BB_G2.AZ_akt := 4714;
   BB_G2.ESH := 504;
   BB_G2.SW_akt := 0.0;
   BB_G2.SW_Auto := 6500.0;
   BB_G2.SW_out := 0.0;
   BB_G3.Status.Bed_vOrt := FALSE;
   BB_G3.Status.Bed_UV := FALSE;
   BB_G3.Status.Bed_NHV := FALSE;
   BB_G3.Status.Bed_PLS := TRUE;
   BB_G3.Status.BA_Hand := FALSE;
   BB_G3.Status.BA_Auto := TRUE;
   BB_G3.Status.RB_Ein1 := FALSE;
   BB_G3.Status.RB_Ein2 := FALSE;
   BB_G3.Status.RB_Aus := TRUE;
   BB_G3.Status.BFR_NS := FALSE;
   BB_G3.Status.BFR_ECS := FALSE;
   BB_G3.Status.BFR_ESK := FALSE;
   BB_G3.Status.BFR_MAZ := FALSE;
   BB_G3.Status.BFR_Rev := FALSE;
   BB_G3.Status.BFR_Ein1 := FALSE;
   BB_G3.Status.BFR_Ein2 := FALSE;
   BB_G3.Status.BM_Ein1 := FALSE;
   BB_G3.Status.BM_Ein2 := FALSE;
   BB_G3.Status.BM_Auf := FALSE;
   BB_G3.Status.BM_Zu := FALSE;
   BB_G3.Status.BM_Ein := FALSE;
   BB_G3.Status.BM_Aus := TRUE;
   BB_G3.Status.BM_Anst1 := FALSE;
   BB_G3.Status.BM_Anst2 := FALSE;
   BB_G3.Status.BM_Auto1 := FALSE;
   BB_G3.Status.BM_Auto2 := FALSE;
   BB_G3.Status.Res_26 := FALSE;
   BB_G3.Status.Res_27 := FALSE;
   BB_G3.Status.BB_NA := TRUE;
   BB_G3.Status.BB_AutoOk := FALSE;
   BB_G3.Status.BB_SS := TRUE;
   BB_G3.Status.BB_SSnq := FALSE;
   BB_G3.Stoerung.St_allg := FALSE;
   BB_G3.Stoerung.St_DMA := FALSE;
   BB_G3.Stoerung.St_DMZ := FALSE;
   BB_G3.Stoerung.St_FU := TRUE;
   BB_G3.Stoerung.St_TL := FALSE;
   BB_G3.Stoerung.St_UDr := FALSE;
   BB_G3.Stoerung.St_UeDr := FALSE;
   BB_G3.Stoerung.St_UeTemp := FALSE;
   BB_G3.Stoerung.St_Leck := FALSE;
   BB_G3.Stoerung.St_UeLM := FALSE;
   BB_G3.Stoerung.St_UeLE := FALSE;
   BB_G3.Stoerung.St_Kom_DP := FALSE;
   BB_G3.Stoerung.St_Kom_int := FALSE;
   BB_G3.Stoerung.St_int := FALSE;
   BB_G3.Stoerung.St_LZ := FALSE;
   BB_G3.Stoerung.St_BefLZ := FALSE;
   BB_G3.Stoerung.Wa_EZ := FALSE;
   BB_G3.Stoerung.Wa_Wart := TRUE;
   BB_G3.Stoerung.St_Strm := FALSE;
   BB_G3.Stoerung.Res_19 := FALSE;
   BB_G3.Stoerung.Res_20 := FALSE;
   BB_G3.Stoerung.Res_21 := FALSE;
   BB_G3.Stoerung.Res_22 := FALSE;
   BB_G3.Stoerung.Res_23 := FALSE;
   BB_G3.Stoerung.Res_24 := FALSE;
   BB_G3.Stoerung.Res_25 := FALSE;
   BB_G3.Stoerung.Res_26 := FALSE;
   BB_G3.Stoerung.Res_27 := FALSE;
   BB_G3.Stoerung.Res_28 := FALSE;
   BB_G3.Stoerung.Res_29 := FALSE;
   BB_G3.Stoerung.Res_30 := FALSE;
   BB_G3.Stoerung.Res_31 := FALSE;
   BB_G3.MW_I := 0.0;
   BB_G3.MW_P := 0.0;
   BB_G3.EZ := 0;
   BB_G3.BZ_akt := 26;
   BB_G3.BZ_ges := 326911;
   BB_G3.AZ_akt := 1226;
   BB_G3.ESH := 366;
   BB_G3.SW_akt := 0.0;
   BB_G3.SW_Auto := 6500.0;
   BB_G3.SW_out := 0.0;
   BB_SHL_G1.Status.Bed_vOrt := FALSE;
   BB_SHL_G1.Status.Bed_UV := FALSE;
   BB_SHL_G1.Status.Bed_NHV := TRUE;
   BB_SHL_G1.Status.Bed_PLS := FALSE;
   BB_SHL_G1.Status.BA_Hand := FALSE;
   BB_SHL_G1.Status.BA_Auto := TRUE;
   BB_SHL_G1.Status.RB_Ein1 := TRUE;
   BB_SHL_G1.Status.RB_Ein2 := FALSE;
   BB_SHL_G1.Status.RB_Aus := FALSE;
   BB_SHL_G1.Status.BFR_NS := FALSE;
   BB_SHL_G1.Status.BFR_ECS := FALSE;
   BB_SHL_G1.Status.BFR_ESK := FALSE;
   BB_SHL_G1.Status.BFR_MAZ := FALSE;
   BB_SHL_G1.Status.BFR_Rev := FALSE;
   BB_SHL_G1.Status.BFR_Ein1 := FALSE;
   BB_SHL_G1.Status.BFR_Ein2 := FALSE;
   BB_SHL_G1.Status.BM_Ein1 := TRUE;
   BB_SHL_G1.Status.BM_Ein2 := FALSE;
   BB_SHL_G1.Status.BM_Auf := FALSE;
   BB_SHL_G1.Status.BM_Zu := FALSE;
   BB_SHL_G1.Status.BM_Ein := TRUE;
   BB_SHL_G1.Status.BM_Aus := FALSE;
   BB_SHL_G1.Status.BM_Anst1 := FALSE;
   BB_SHL_G1.Status.BM_Anst2 := FALSE;
   BB_SHL_G1.Status.BM_Auto1 := FALSE;
   BB_SHL_G1.Status.BM_Auto2 := FALSE;
   BB_SHL_G1.Status.Res_26 := FALSE;
   BB_SHL_G1.Status.Res_27 := FALSE;
   BB_SHL_G1.Status.BB_NA := FALSE;
   BB_SHL_G1.Status.BB_AutoOk := TRUE;
   BB_SHL_G1.Status.BB_SS := FALSE;
   BB_SHL_G1.Status.BB_SSnq := FALSE;
   BB_SHL_G1.Stoerung.St_allg := FALSE;
   BB_SHL_G1.Stoerung.St_DMA := FALSE;
   BB_SHL_G1.Stoerung.St_DMZ := FALSE;
   BB_SHL_G1.Stoerung.St_FU := FALSE;
   BB_SHL_G1.Stoerung.St_TL := FALSE;
   BB_SHL_G1.Stoerung.St_UDr := FALSE;
   BB_SHL_G1.Stoerung.St_UeDr := FALSE;
   BB_SHL_G1.Stoerung.St_UeTemp := FALSE;
   BB_SHL_G1.Stoerung.St_Leck := FALSE;
   BB_SHL_G1.Stoerung.St_UeLM := FALSE;
   BB_SHL_G1.Stoerung.St_UeLE := FALSE;
   BB_SHL_G1.Stoerung.St_Kom_DP := FALSE;
   BB_SHL_G1.Stoerung.St_Kom_int := FALSE;
   BB_SHL_G1.Stoerung.St_int := FALSE;
   BB_SHL_G1.Stoerung.St_LZ := FALSE;
   BB_SHL_G1.Stoerung.St_BefLZ := FALSE;
   BB_SHL_G1.Stoerung.Wa_EZ := FALSE;
   BB_SHL_G1.Stoerung.Wa_Wart := FALSE;
   BB_SHL_G1.Stoerung.St_Strm := FALSE;
   BB_SHL_G1.Stoerung.Res_19 := FALSE;
   BB_SHL_G1.Stoerung.Res_20 := FALSE;
   BB_SHL_G1.Stoerung.Res_21 := FALSE;
   BB_SHL_G1.Stoerung.Res_22 := FALSE;
   BB_SHL_G1.Stoerung.Res_23 := FALSE;
   BB_SHL_G1.Stoerung.Res_24 := FALSE;
   BB_SHL_G1.Stoerung.Res_25 := FALSE;
   BB_SHL_G1.Stoerung.Res_26 := FALSE;
   BB_SHL_G1.Stoerung.Res_27 := FALSE;
   BB_SHL_G1.Stoerung.Res_28 := FALSE;
   BB_SHL_G1.Stoerung.Res_29 := FALSE;
   BB_SHL_G1.Stoerung.Res_30 := FALSE;
   BB_SHL_G1.Stoerung.Res_31 := FALSE;
   BB_SHL_G1.MW_I := 0.0;
   BB_SHL_G1.MW_P := 0.0;
   BB_SHL_G1.EZ := 0;
   BB_SHL_G1.BZ_akt := 989;
   BB_SHL_G1.BZ_ges := 49708252;
   BB_SHL_G1.AZ_akt := 884;
   BB_SHL_G1.ESH := 35991;
   BB_SHL_G1.SW_akt := 0.0;
   BB_SHL_G1.SW_Auto := 0.0;
   BB_SHL_G1.SW_out := 0.0;
   BB_SHL_G2.Status.Bed_vOrt := FALSE;
   BB_SHL_G2.Status.Bed_UV := FALSE;
   BB_SHL_G2.Status.Bed_NHV := TRUE;
   BB_SHL_G2.Status.Bed_PLS := FALSE;
   BB_SHL_G2.Status.BA_Hand := FALSE;
   BB_SHL_G2.Status.BA_Auto := TRUE;
   BB_SHL_G2.Status.RB_Ein1 := FALSE;
   BB_SHL_G2.Status.RB_Ein2 := FALSE;
   BB_SHL_G2.Status.RB_Aus := TRUE;
   BB_SHL_G2.Status.BFR_NS := FALSE;
   BB_SHL_G2.Status.BFR_ECS := FALSE;
   BB_SHL_G2.Status.BFR_ESK := FALSE;
   BB_SHL_G2.Status.BFR_MAZ := FALSE;
   BB_SHL_G2.Status.BFR_Rev := FALSE;
   BB_SHL_G2.Status.BFR_Ein1 := FALSE;
   BB_SHL_G2.Status.BFR_Ein2 := FALSE;
   BB_SHL_G2.Status.BM_Ein1 := FALSE;
   BB_SHL_G2.Status.BM_Ein2 := FALSE;
   BB_SHL_G2.Status.BM_Auf := FALSE;
   BB_SHL_G2.Status.BM_Zu := FALSE;
   BB_SHL_G2.Status.BM_Ein := FALSE;
   BB_SHL_G2.Status.BM_Aus := TRUE;
   BB_SHL_G2.Status.BM_Anst1 := FALSE;
   BB_SHL_G2.Status.BM_Anst2 := FALSE;
   BB_SHL_G2.Status.BM_Auto1 := FALSE;
   BB_SHL_G2.Status.BM_Auto2 := FALSE;
   BB_SHL_G2.Status.Res_26 := FALSE;
   BB_SHL_G2.Status.Res_27 := FALSE;
   BB_SHL_G2.Status.BB_NA := FALSE;
   BB_SHL_G2.Status.BB_AutoOk := TRUE;
   BB_SHL_G2.Status.BB_SS := FALSE;
   BB_SHL_G2.Status.BB_SSnq := FALSE;
   BB_SHL_G2.Stoerung.St_allg := FALSE;
   BB_SHL_G2.Stoerung.St_DMA := FALSE;
   BB_SHL_G2.Stoerung.St_DMZ := FALSE;
   BB_SHL_G2.Stoerung.St_FU := FALSE;
   BB_SHL_G2.Stoerung.St_TL := FALSE;
   BB_SHL_G2.Stoerung.St_UDr := FALSE;
   BB_SHL_G2.Stoerung.St_UeDr := FALSE;
   BB_SHL_G2.Stoerung.St_UeTemp := FALSE;
   BB_SHL_G2.Stoerung.St_Leck := FALSE;
   BB_SHL_G2.Stoerung.St_UeLM := FALSE;
   BB_SHL_G2.Stoerung.St_UeLE := FALSE;
   BB_SHL_G2.Stoerung.St_Kom_DP := FALSE;
   BB_SHL_G2.Stoerung.St_Kom_int := FALSE;
   BB_SHL_G2.Stoerung.St_int := FALSE;
   BB_SHL_G2.Stoerung.St_LZ := FALSE;
   BB_SHL_G2.Stoerung.St_BefLZ := FALSE;
   BB_SHL_G2.Stoerung.Wa_EZ := FALSE;
   BB_SHL_G2.Stoerung.Wa_Wart := FALSE;
   BB_SHL_G2.Stoerung.St_Strm := FALSE;
   BB_SHL_G2.Stoerung.Res_19 := FALSE;
   BB_SHL_G2.Stoerung.Res_20 := FALSE;
   BB_SHL_G2.Stoerung.Res_21 := FALSE;
   BB_SHL_G2.Stoerung.Res_22 := FALSE;
   BB_SHL_G2.Stoerung.Res_23 := FALSE;
   BB_SHL_G2.Stoerung.Res_24 := FALSE;
   BB_SHL_G2.Stoerung.Res_25 := FALSE;
   BB_SHL_G2.Stoerung.Res_26 := FALSE;
   BB_SHL_G2.Stoerung.Res_27 := FALSE;
   BB_SHL_G2.Stoerung.Res_28 := FALSE;
   BB_SHL_G2.Stoerung.Res_29 := FALSE;
   BB_SHL_G2.Stoerung.Res_30 := FALSE;
   BB_SHL_G2.Stoerung.Res_31 := FALSE;
   BB_SHL_G2.MW_I := 0.0;
   BB_SHL_G2.MW_P := 0.0;
   BB_SHL_G2.EZ := 0;
   BB_SHL_G2.BZ_akt := 634;
   BB_SHL_G2.BZ_ges := 62823119;
   BB_SHL_G2.AZ_akt := 4170;
   BB_SHL_G2.ESH := 32997;
   BB_SHL_G2.SW_akt := 0.0;
   BB_SHL_G2.SW_Auto := 0.0;
   BB_SHL_G2.SW_out := 0.0;
   BB_SHL_G3.Status.Bed_vOrt := FALSE;
   BB_SHL_G3.Status.Bed_UV := FALSE;
   BB_SHL_G3.Status.Bed_NHV := TRUE;
   BB_SHL_G3.Status.Bed_PLS := FALSE;
   BB_SHL_G3.Status.BA_Hand := FALSE;
   BB_SHL_G3.Status.BA_Auto := TRUE;
   BB_SHL_G3.Status.RB_Ein1 := FALSE;
   BB_SHL_G3.Status.RB_Ein2 := FALSE;
   BB_SHL_G3.Status.RB_Aus := TRUE;
   BB_SHL_G3.Status.BFR_NS := FALSE;
   BB_SHL_G3.Status.BFR_ECS := FALSE;
   BB_SHL_G3.Status.BFR_ESK := FALSE;
   BB_SHL_G3.Status.BFR_MAZ := FALSE;
   BB_SHL_G3.Status.BFR_Rev := FALSE;
   BB_SHL_G3.Status.BFR_Ein1 := FALSE;
   BB_SHL_G3.Status.BFR_Ein2 := FALSE;
   BB_SHL_G3.Status.BM_Ein1 := FALSE;
   BB_SHL_G3.Status.BM_Ein2 := FALSE;
   BB_SHL_G3.Status.BM_Auf := FALSE;
   BB_SHL_G3.Status.BM_Zu := FALSE;
   BB_SHL_G3.Status.BM_Ein := FALSE;
   BB_SHL_G3.Status.BM_Aus := TRUE;
   BB_SHL_G3.Status.BM_Anst1 := FALSE;
   BB_SHL_G3.Status.BM_Anst2 := FALSE;
   BB_SHL_G3.Status.BM_Auto1 := FALSE;
   BB_SHL_G3.Status.BM_Auto2 := FALSE;
   BB_SHL_G3.Status.Res_26 := FALSE;
   BB_SHL_G3.Status.Res_27 := FALSE;
   BB_SHL_G3.Status.BB_NA := FALSE;
   BB_SHL_G3.Status.BB_AutoOk := TRUE;
   BB_SHL_G3.Status.BB_SS := FALSE;
   BB_SHL_G3.Status.BB_SSnq := FALSE;
   BB_SHL_G3.Stoerung.St_allg := FALSE;
   BB_SHL_G3.Stoerung.St_DMA := FALSE;
   BB_SHL_G3.Stoerung.St_DMZ := FALSE;
   BB_SHL_G3.Stoerung.St_FU := FALSE;
   BB_SHL_G3.Stoerung.St_TL := FALSE;
   BB_SHL_G3.Stoerung.St_UDr := FALSE;
   BB_SHL_G3.Stoerung.St_UeDr := FALSE;
   BB_SHL_G3.Stoerung.St_UeTemp := FALSE;
   BB_SHL_G3.Stoerung.St_Leck := FALSE;
   BB_SHL_G3.Stoerung.St_UeLM := FALSE;
   BB_SHL_G3.Stoerung.St_UeLE := FALSE;
   BB_SHL_G3.Stoerung.St_Kom_DP := FALSE;
   BB_SHL_G3.Stoerung.St_Kom_int := FALSE;
   BB_SHL_G3.Stoerung.St_int := FALSE;
   BB_SHL_G3.Stoerung.St_LZ := FALSE;
   BB_SHL_G3.Stoerung.St_BefLZ := FALSE;
   BB_SHL_G3.Stoerung.Wa_EZ := FALSE;
   BB_SHL_G3.Stoerung.Wa_Wart := FALSE;
   BB_SHL_G3.Stoerung.St_Strm := FALSE;
   BB_SHL_G3.Stoerung.Res_19 := FALSE;
   BB_SHL_G3.Stoerung.Res_20 := FALSE;
   BB_SHL_G3.Stoerung.Res_21 := FALSE;
   BB_SHL_G3.Stoerung.Res_22 := FALSE;
   BB_SHL_G3.Stoerung.Res_23 := FALSE;
   BB_SHL_G3.Stoerung.Res_24 := FALSE;
   BB_SHL_G3.Stoerung.Res_25 := FALSE;
   BB_SHL_G3.Stoerung.Res_26 := FALSE;
   BB_SHL_G3.Stoerung.Res_27 := FALSE;
   BB_SHL_G3.Stoerung.Res_28 := FALSE;
   BB_SHL_G3.Stoerung.Res_29 := FALSE;
   BB_SHL_G3.Stoerung.Res_30 := FALSE;
   BB_SHL_G3.Stoerung.Res_31 := FALSE;
   BB_SHL_G3.MW_I := 0.0;
   BB_SHL_G3.MW_P := 0.0;
   BB_SHL_G3.EZ := 0;
   BB_SHL_G3.BZ_akt := 601;
   BB_SHL_G3.BZ_ges := 59909177;
   BB_SHL_G3.AZ_akt := 654;
   BB_SHL_G3.ESH := 30786;
   BB_SHL_G3.SW_akt := 0.0;
   BB_SHL_G3.SW_Auto := 0.0;
   BB_SHL_G3.SW_out := 0.0;
   BB_AV.Status.Bed_vOrt := FALSE;
   BB_AV.Status.Bed_UV := FALSE;
   BB_AV.Status.Bed_NHV := TRUE;
   BB_AV.Status.Bed_PLS := FALSE;
   BB_AV.Status.BA_Hand := FALSE;
   BB_AV.Status.BA_Auto := TRUE;
   BB_AV.Status.RB_Ein1 := FALSE;
   BB_AV.Status.RB_Ein2 := FALSE;
   BB_AV.Status.RB_Aus := TRUE;
   BB_AV.Status.BFR_NS := FALSE;
   BB_AV.Status.BFR_ECS := FALSE;
   BB_AV.Status.BFR_ESK := FALSE;
   BB_AV.Status.BFR_MAZ := FALSE;
   BB_AV.Status.BFR_Rev := FALSE;
   BB_AV.Status.BFR_Ein1 := FALSE;
   BB_AV.Status.BFR_Ein2 := FALSE;
   BB_AV.Status.BM_Ein1 := FALSE;
   BB_AV.Status.BM_Ein2 := FALSE;
   BB_AV.Status.BM_Auf := FALSE;
   BB_AV.Status.BM_Zu := FALSE;
   BB_AV.Status.BM_Ein := FALSE;
   BB_AV.Status.BM_Aus := TRUE;
   BB_AV.Status.BM_Anst1 := FALSE;
   BB_AV.Status.BM_Anst2 := FALSE;
   BB_AV.Status.BM_Auto1 := FALSE;
   BB_AV.Status.BM_Auto2 := FALSE;
   BB_AV.Status.Res_26 := FALSE;
   BB_AV.Status.Res_27 := FALSE;
   BB_AV.Status.BB_NA := FALSE;
   BB_AV.Status.BB_AutoOk := TRUE;
   BB_AV.Status.BB_SS := FALSE;
   BB_AV.Status.BB_SSnq := FALSE;
   BB_AV.Stoerung.St_allg := FALSE;
   BB_AV.Stoerung.St_DMA := FALSE;
   BB_AV.Stoerung.St_DMZ := FALSE;
   BB_AV.Stoerung.St_FU := FALSE;
   BB_AV.Stoerung.St_TL := FALSE;
   BB_AV.Stoerung.St_UDr := FALSE;
   BB_AV.Stoerung.St_UeDr := FALSE;
   BB_AV.Stoerung.St_UeTemp := FALSE;
   BB_AV.Stoerung.St_Leck := FALSE;
   BB_AV.Stoerung.St_UeLM := FALSE;
   BB_AV.Stoerung.St_UeLE := FALSE;
   BB_AV.Stoerung.St_Kom_DP := FALSE;
   BB_AV.Stoerung.St_Kom_int := FALSE;
   BB_AV.Stoerung.St_int := FALSE;
   BB_AV.Stoerung.St_LZ := FALSE;
   BB_AV.Stoerung.St_BefLZ := FALSE;
   BB_AV.Stoerung.Wa_EZ := FALSE;
   BB_AV.Stoerung.Wa_Wart := FALSE;
   BB_AV.Stoerung.St_Strm := FALSE;
   BB_AV.Stoerung.Res_19 := FALSE;
   BB_AV.Stoerung.Res_20 := FALSE;
   BB_AV.Stoerung.Res_21 := FALSE;
   BB_AV.Stoerung.Res_22 := FALSE;
   BB_AV.Stoerung.Res_23 := FALSE;
   BB_AV.Stoerung.Res_24 := FALSE;
   BB_AV.Stoerung.Res_25 := FALSE;
   BB_AV.Stoerung.Res_26 := FALSE;
   BB_AV.Stoerung.Res_27 := FALSE;
   BB_AV.Stoerung.Res_28 := FALSE;
   BB_AV.Stoerung.Res_29 := FALSE;
   BB_AV.Stoerung.Res_30 := FALSE;
   BB_AV.Stoerung.Res_31 := FALSE;
   BB_AV.MW_I := 0.0;
   BB_AV.MW_P := 0.0;
   BB_AV.EZ := 0;
   BB_AV.BZ_akt := 165;
   BB_AV.BZ_ges := 6353798;
   BB_AV.AZ_akt := 17356664;
   BB_AV.ESH := 1654;
   BB_AV.SW_akt := 0.0;
   BB_AV.SW_Auto := 0.0;
   BB_AV.SW_out := 0.0;
   BB_LS1.Status.Bed_vOrt := FALSE;
   BB_LS1.Status.Bed_UV := FALSE;
   BB_LS1.Status.Bed_NHV := FALSE;
   BB_LS1.Status.Bed_PLS := TRUE;
   BB_LS1.Status.BA_Hand := FALSE;
   BB_LS1.Status.BA_Auto := TRUE;
   BB_LS1.Status.RB_Ein1 := FALSE;
   BB_LS1.Status.RB_Ein2 := FALSE;
   BB_LS1.Status.RB_Aus := TRUE;
   BB_LS1.Status.BFR_NS := FALSE;
   BB_LS1.Status.BFR_ECS := FALSE;
   BB_LS1.Status.BFR_ESK := FALSE;
   BB_LS1.Status.BFR_MAZ := FALSE;
   BB_LS1.Status.BFR_Rev := FALSE;
   BB_LS1.Status.BFR_Ein1 := FALSE;
   BB_LS1.Status.BFR_Ein2 := FALSE;
   BB_LS1.Status.BM_Ein1 := FALSE;
   BB_LS1.Status.BM_Ein2 := FALSE;
   BB_LS1.Status.BM_Auf := FALSE;
   BB_LS1.Status.BM_Zu := TRUE;
   BB_LS1.Status.BM_Ein := FALSE;
   BB_LS1.Status.BM_Aus := TRUE;
   BB_LS1.Status.BM_Anst1 := FALSE;
   BB_LS1.Status.BM_Anst2 := FALSE;
   BB_LS1.Status.BM_Auto1 := FALSE;
   BB_LS1.Status.BM_Auto2 := TRUE;
   BB_LS1.Status.Res_26 := FALSE;
   BB_LS1.Status.Res_27 := FALSE;
   BB_LS1.Status.BB_NA := FALSE;
   BB_LS1.Status.BB_AutoOk := TRUE;
   BB_LS1.Status.BB_SS := FALSE;
   BB_LS1.Status.BB_SSnq := FALSE;
   BB_LS1.Stoerung.St_allg := FALSE;
   BB_LS1.Stoerung.St_DMA := FALSE;
   BB_LS1.Stoerung.St_DMZ := FALSE;
   BB_LS1.Stoerung.St_FU := FALSE;
   BB_LS1.Stoerung.St_TL := FALSE;
   BB_LS1.Stoerung.St_UDr := FALSE;
   BB_LS1.Stoerung.St_UeDr := FALSE;
   BB_LS1.Stoerung.St_UeTemp := FALSE;
   BB_LS1.Stoerung.St_Leck := FALSE;
   BB_LS1.Stoerung.St_UeLM := FALSE;
   BB_LS1.Stoerung.St_UeLE := FALSE;
   BB_LS1.Stoerung.St_Kom_DP := FALSE;
   BB_LS1.Stoerung.St_Kom_int := FALSE;
   BB_LS1.Stoerung.St_int := FALSE;
   BB_LS1.Stoerung.St_LZ := FALSE;
   BB_LS1.Stoerung.St_BefLZ := FALSE;
   BB_LS1.Stoerung.Wa_EZ := FALSE;
   BB_LS1.Stoerung.Wa_Wart := FALSE;
   BB_LS1.Stoerung.St_Strm := FALSE;
   BB_LS1.Stoerung.Res_19 := FALSE;
   BB_LS1.Stoerung.Res_20 := FALSE;
   BB_LS1.Stoerung.Res_21 := FALSE;
   BB_LS1.Stoerung.Res_22 := FALSE;
   BB_LS1.Stoerung.Res_23 := FALSE;
   BB_LS1.Stoerung.Res_24 := FALSE;
   BB_LS1.Stoerung.Res_25 := FALSE;
   BB_LS1.Stoerung.Res_26 := FALSE;
   BB_LS1.Stoerung.Res_27 := FALSE;
   BB_LS1.Stoerung.Res_28 := FALSE;
   BB_LS1.Stoerung.Res_29 := FALSE;
   BB_LS1.Stoerung.Res_30 := FALSE;
   BB_LS1.Stoerung.Res_31 := FALSE;
   BB_LS1.MW_I := 0.0;
   BB_LS1.MW_P := 0.0;
   BB_LS1.EZ := 0;
   BB_LS1.BZ_akt := 51;
   BB_LS1.BZ_ges := 35061;
   BB_LS1.AZ_akt := 3998;
   BB_LS1.ESH := 1165;
   BB_LS1.SW_akt := 0.0;
   BB_LS1.SW_Auto := 0.0;
   BB_LS1.SW_out := 0.0;
   BB_LS2.Status.Bed_vOrt := FALSE;
   BB_LS2.Status.Bed_UV := FALSE;
   BB_LS2.Status.Bed_NHV := FALSE;
   BB_LS2.Status.Bed_PLS := TRUE;
   BB_LS2.Status.BA_Hand := TRUE;
   BB_LS2.Status.BA_Auto := FALSE;
   BB_LS2.Status.RB_Ein1 := FALSE;
   BB_LS2.Status.RB_Ein2 := FALSE;
   BB_LS2.Status.RB_Aus := TRUE;
   BB_LS2.Status.BFR_NS := FALSE;
   BB_LS2.Status.BFR_ECS := FALSE;
   BB_LS2.Status.BFR_ESK := FALSE;
   BB_LS2.Status.BFR_MAZ := FALSE;
   BB_LS2.Status.BFR_Rev := FALSE;
   BB_LS2.Status.BFR_Ein1 := FALSE;
   BB_LS2.Status.BFR_Ein2 := FALSE;
   BB_LS2.Status.BM_Ein1 := FALSE;
   BB_LS2.Status.BM_Ein2 := FALSE;
   BB_LS2.Status.BM_Auf := TRUE;
   BB_LS2.Status.BM_Zu := FALSE;
   BB_LS2.Status.BM_Ein := FALSE;
   BB_LS2.Status.BM_Aus := TRUE;
   BB_LS2.Status.BM_Anst1 := FALSE;
   BB_LS2.Status.BM_Anst2 := FALSE;
   BB_LS2.Status.BM_Auto1 := FALSE;
   BB_LS2.Status.BM_Auto2 := TRUE;
   BB_LS2.Status.Res_26 := FALSE;
   BB_LS2.Status.Res_27 := FALSE;
   BB_LS2.Status.BB_NA := FALSE;
   BB_LS2.Status.BB_AutoOk := FALSE;
   BB_LS2.Status.BB_SS := FALSE;
   BB_LS2.Status.BB_SSnq := FALSE;
   BB_LS2.Stoerung.St_allg := FALSE;
   BB_LS2.Stoerung.St_DMA := FALSE;
   BB_LS2.Stoerung.St_DMZ := FALSE;
   BB_LS2.Stoerung.St_FU := FALSE;
   BB_LS2.Stoerung.St_TL := FALSE;
   BB_LS2.Stoerung.St_UDr := FALSE;
   BB_LS2.Stoerung.St_UeDr := FALSE;
   BB_LS2.Stoerung.St_UeTemp := FALSE;
   BB_LS2.Stoerung.St_Leck := FALSE;
   BB_LS2.Stoerung.St_UeLM := FALSE;
   BB_LS2.Stoerung.St_UeLE := FALSE;
   BB_LS2.Stoerung.St_Kom_DP := FALSE;
   BB_LS2.Stoerung.St_Kom_int := FALSE;
   BB_LS2.Stoerung.St_int := FALSE;
   BB_LS2.Stoerung.St_LZ := FALSE;
   BB_LS2.Stoerung.St_BefLZ := FALSE;
   BB_LS2.Stoerung.Wa_EZ := FALSE;
   BB_LS2.Stoerung.Wa_Wart := FALSE;
   BB_LS2.Stoerung.St_Strm := FALSE;
   BB_LS2.Stoerung.Res_19 := FALSE;
   BB_LS2.Stoerung.Res_20 := FALSE;
   BB_LS2.Stoerung.Res_21 := FALSE;
   BB_LS2.Stoerung.Res_22 := FALSE;
   BB_LS2.Stoerung.Res_23 := FALSE;
   BB_LS2.Stoerung.Res_24 := FALSE;
   BB_LS2.Stoerung.Res_25 := FALSE;
   BB_LS2.Stoerung.Res_26 := FALSE;
   BB_LS2.Stoerung.Res_27 := FALSE;
   BB_LS2.Stoerung.Res_28 := FALSE;
   BB_LS2.Stoerung.Res_29 := FALSE;
   BB_LS2.Stoerung.Res_30 := FALSE;
   BB_LS2.Stoerung.Res_31 := FALSE;
   BB_LS2.MW_I := 0.0;
   BB_LS2.MW_P := 0.0;
   BB_LS2.EZ := 0;
   BB_LS2.BZ_akt := 30;
   BB_LS2.BZ_ges := 33042;
   BB_LS2.AZ_akt := 1192;
   BB_LS2.ESH := 1074;
   BB_LS2.SW_akt := 0.0;
   BB_LS2.SW_Auto := 0.0;
   BB_LS2.SW_out := 0.0;
   BB1_RZP1.Status.Bed_vOrt := FALSE;
   BB1_RZP1.Status.Bed_UV := FALSE;
   BB1_RZP1.Status.Bed_NHV := FALSE;
   BB1_RZP1.Status.Bed_PLS := TRUE;
   BB1_RZP1.Status.BA_Hand := FALSE;
   BB1_RZP1.Status.BA_Auto := TRUE;
   BB1_RZP1.Status.RB_Ein1 := FALSE;
   BB1_RZP1.Status.RB_Ein2 := FALSE;
   BB1_RZP1.Status.RB_Aus := TRUE;
   BB1_RZP1.Status.BFR_NS := FALSE;
   BB1_RZP1.Status.BFR_ECS := FALSE;
   BB1_RZP1.Status.BFR_ESK := FALSE;
   BB1_RZP1.Status.BFR_MAZ := FALSE;
   BB1_RZP1.Status.BFR_Rev := FALSE;
   BB1_RZP1.Status.BFR_Ein1 := FALSE;
   BB1_RZP1.Status.BFR_Ein2 := FALSE;
   BB1_RZP1.Status.BM_Ein1 := FALSE;
   BB1_RZP1.Status.BM_Ein2 := FALSE;
   BB1_RZP1.Status.BM_Auf := FALSE;
   BB1_RZP1.Status.BM_Zu := FALSE;
   BB1_RZP1.Status.BM_Ein := FALSE;
   BB1_RZP1.Status.BM_Aus := TRUE;
   BB1_RZP1.Status.BM_Anst1 := FALSE;
   BB1_RZP1.Status.BM_Anst2 := FALSE;
   BB1_RZP1.Status.BM_Auto1 := FALSE;
   BB1_RZP1.Status.BM_Auto2 := FALSE;
   BB1_RZP1.Status.Res_26 := FALSE;
   BB1_RZP1.Status.Res_27 := FALSE;
   BB1_RZP1.Status.BB_NA := FALSE;
   BB1_RZP1.Status.BB_AutoOk := TRUE;
   BB1_RZP1.Status.BB_SS := FALSE;
   BB1_RZP1.Status.BB_SSnq := FALSE;
   BB1_RZP1.Stoerung.St_allg := FALSE;
   BB1_RZP1.Stoerung.St_DMA := FALSE;
   BB1_RZP1.Stoerung.St_DMZ := FALSE;
   BB1_RZP1.Stoerung.St_FU := FALSE;
   BB1_RZP1.Stoerung.St_TL := FALSE;
   BB1_RZP1.Stoerung.St_UDr := FALSE;
   BB1_RZP1.Stoerung.St_UeDr := FALSE;
   BB1_RZP1.Stoerung.St_UeTemp := FALSE;
   BB1_RZP1.Stoerung.St_Leck := FALSE;
   BB1_RZP1.Stoerung.St_UeLM := FALSE;
   BB1_RZP1.Stoerung.St_UeLE := FALSE;
   BB1_RZP1.Stoerung.St_Kom_DP := FALSE;
   BB1_RZP1.Stoerung.St_Kom_int := FALSE;
   BB1_RZP1.Stoerung.St_int := FALSE;
   BB1_RZP1.Stoerung.St_LZ := FALSE;
   BB1_RZP1.Stoerung.St_BefLZ := FALSE;
   BB1_RZP1.Stoerung.Wa_EZ := FALSE;
   BB1_RZP1.Stoerung.Wa_Wart := FALSE;
   BB1_RZP1.Stoerung.St_Strm := FALSE;
   BB1_RZP1.Stoerung.Res_19 := FALSE;
   BB1_RZP1.Stoerung.Res_20 := FALSE;
   BB1_RZP1.Stoerung.Res_21 := FALSE;
   BB1_RZP1.Stoerung.Res_22 := FALSE;
   BB1_RZP1.Stoerung.Res_23 := FALSE;
   BB1_RZP1.Stoerung.Res_24 := FALSE;
   BB1_RZP1.Stoerung.Res_25 := FALSE;
   BB1_RZP1.Stoerung.Res_26 := FALSE;
   BB1_RZP1.Stoerung.Res_27 := FALSE;
   BB1_RZP1.Stoerung.Res_28 := FALSE;
   BB1_RZP1.Stoerung.Res_29 := FALSE;
   BB1_RZP1.Stoerung.Res_30 := FALSE;
   BB1_RZP1.Stoerung.Res_31 := FALSE;
   BB1_RZP1.MW_I := 0.0;
   BB1_RZP1.MW_P := 0.0;
   BB1_RZP1.EZ := 0;
   BB1_RZP1.BZ_akt := 861;
   BB1_RZP1.BZ_ges := 115348;
   BB1_RZP1.AZ_akt := 4714;
   BB1_RZP1.ESH := 134;
   BB1_RZP1.SW_akt := 0.0;
   BB1_RZP1.SW_Auto := 0.0;
   BB1_RZP1.SW_out := 0.0;
   BB1_RZP2.Status.Bed_vOrt := FALSE;
   BB1_RZP2.Status.Bed_UV := FALSE;
   BB1_RZP2.Status.Bed_NHV := FALSE;
   BB1_RZP2.Status.Bed_PLS := TRUE;
   BB1_RZP2.Status.BA_Hand := FALSE;
   BB1_RZP2.Status.BA_Auto := TRUE;
   BB1_RZP2.Status.RB_Ein1 := FALSE;
   BB1_RZP2.Status.RB_Ein2 := FALSE;
   BB1_RZP2.Status.RB_Aus := TRUE;
   BB1_RZP2.Status.BFR_NS := FALSE;
   BB1_RZP2.Status.BFR_ECS := FALSE;
   BB1_RZP2.Status.BFR_ESK := FALSE;
   BB1_RZP2.Status.BFR_MAZ := FALSE;
   BB1_RZP2.Status.BFR_Rev := FALSE;
   BB1_RZP2.Status.BFR_Ein1 := FALSE;
   BB1_RZP2.Status.BFR_Ein2 := FALSE;
   BB1_RZP2.Status.BM_Ein1 := FALSE;
   BB1_RZP2.Status.BM_Ein2 := FALSE;
   BB1_RZP2.Status.BM_Auf := FALSE;
   BB1_RZP2.Status.BM_Zu := FALSE;
   BB1_RZP2.Status.BM_Ein := FALSE;
   BB1_RZP2.Status.BM_Aus := TRUE;
   BB1_RZP2.Status.BM_Anst1 := FALSE;
   BB1_RZP2.Status.BM_Anst2 := FALSE;
   BB1_RZP2.Status.BM_Auto1 := FALSE;
   BB1_RZP2.Status.BM_Auto2 := FALSE;
   BB1_RZP2.Status.Res_26 := FALSE;
   BB1_RZP2.Status.Res_27 := FALSE;
   BB1_RZP2.Status.BB_NA := FALSE;
   BB1_RZP2.Status.BB_AutoOk := TRUE;
   BB1_RZP2.Status.BB_SS := FALSE;
   BB1_RZP2.Status.BB_SSnq := FALSE;
   BB1_RZP2.Stoerung.St_allg := FALSE;
   BB1_RZP2.Stoerung.St_DMA := FALSE;
   BB1_RZP2.Stoerung.St_DMZ := FALSE;
   BB1_RZP2.Stoerung.St_FU := FALSE;
   BB1_RZP2.Stoerung.St_TL := FALSE;
   BB1_RZP2.Stoerung.St_UDr := FALSE;
   BB1_RZP2.Stoerung.St_UeDr := FALSE;
   BB1_RZP2.Stoerung.St_UeTemp := FALSE;
   BB1_RZP2.Stoerung.St_Leck := FALSE;
   BB1_RZP2.Stoerung.St_UeLM := FALSE;
   BB1_RZP2.Stoerung.St_UeLE := FALSE;
   BB1_RZP2.Stoerung.St_Kom_DP := FALSE;
   BB1_RZP2.Stoerung.St_Kom_int := FALSE;
   BB1_RZP2.Stoerung.St_int := FALSE;
   BB1_RZP2.Stoerung.St_LZ := FALSE;
   BB1_RZP2.Stoerung.St_BefLZ := FALSE;
   BB1_RZP2.Stoerung.Wa_EZ := FALSE;
   BB1_RZP2.Stoerung.Wa_Wart := FALSE;
   BB1_RZP2.Stoerung.St_Strm := FALSE;
   BB1_RZP2.Stoerung.Res_19 := FALSE;
   BB1_RZP2.Stoerung.Res_20 := FALSE;
   BB1_RZP2.Stoerung.Res_21 := FALSE;
   BB1_RZP2.Stoerung.Res_22 := FALSE;
   BB1_RZP2.Stoerung.Res_23 := FALSE;
   BB1_RZP2.Stoerung.Res_24 := FALSE;
   BB1_RZP2.Stoerung.Res_25 := FALSE;
   BB1_RZP2.Stoerung.Res_26 := FALSE;
   BB1_RZP2.Stoerung.Res_27 := FALSE;
   BB1_RZP2.Stoerung.Res_28 := FALSE;
   BB1_RZP2.Stoerung.Res_29 := FALSE;
   BB1_RZP2.Stoerung.Res_30 := FALSE;
   BB1_RZP2.Stoerung.Res_31 := FALSE;
   BB1_RZP2.MW_I := 0.0;
   BB1_RZP2.MW_P := 0.0;
   BB1_RZP2.EZ := 0;
   BB1_RZP2.BZ_akt := 860;
   BB1_RZP2.BZ_ges := 116200;
   BB1_RZP2.AZ_akt := 1286;
   BB1_RZP2.ESH := 135;
   BB1_RZP2.SW_akt := 0.0;
   BB1_RZP2.SW_Auto := 0.0;
   BB1_RZP2.SW_out := 0.0;
   BB1_UeSP.Status.Bed_vOrt := FALSE;
   BB1_UeSP.Status.Bed_UV := FALSE;
   BB1_UeSP.Status.Bed_NHV := FALSE;
   BB1_UeSP.Status.Bed_PLS := TRUE;
   BB1_UeSP.Status.BA_Hand := FALSE;
   BB1_UeSP.Status.BA_Auto := TRUE;
   BB1_UeSP.Status.RB_Ein1 := FALSE;
   BB1_UeSP.Status.RB_Ein2 := FALSE;
   BB1_UeSP.Status.RB_Aus := TRUE;
   BB1_UeSP.Status.BFR_NS := FALSE;
   BB1_UeSP.Status.BFR_ECS := FALSE;
   BB1_UeSP.Status.BFR_ESK := FALSE;
   BB1_UeSP.Status.BFR_MAZ := FALSE;
   BB1_UeSP.Status.BFR_Rev := FALSE;
   BB1_UeSP.Status.BFR_Ein1 := FALSE;
   BB1_UeSP.Status.BFR_Ein2 := FALSE;
   BB1_UeSP.Status.BM_Ein1 := FALSE;
   BB1_UeSP.Status.BM_Ein2 := FALSE;
   BB1_UeSP.Status.BM_Auf := FALSE;
   BB1_UeSP.Status.BM_Zu := FALSE;
   BB1_UeSP.Status.BM_Ein := FALSE;
   BB1_UeSP.Status.BM_Aus := TRUE;
   BB1_UeSP.Status.BM_Anst1 := FALSE;
   BB1_UeSP.Status.BM_Anst2 := FALSE;
   BB1_UeSP.Status.BM_Auto1 := FALSE;
   BB1_UeSP.Status.BM_Auto2 := FALSE;
   BB1_UeSP.Status.Res_26 := FALSE;
   BB1_UeSP.Status.Res_27 := FALSE;
   BB1_UeSP.Status.BB_NA := FALSE;
   BB1_UeSP.Status.BB_AutoOk := TRUE;
   BB1_UeSP.Status.BB_SS := FALSE;
   BB1_UeSP.Status.BB_SSnq := FALSE;
   BB1_UeSP.Stoerung.St_allg := FALSE;
   BB1_UeSP.Stoerung.St_DMA := FALSE;
   BB1_UeSP.Stoerung.St_DMZ := FALSE;
   BB1_UeSP.Stoerung.St_FU := FALSE;
   BB1_UeSP.Stoerung.St_TL := FALSE;
   BB1_UeSP.Stoerung.St_UDr := FALSE;
   BB1_UeSP.Stoerung.St_UeDr := FALSE;
   BB1_UeSP.Stoerung.St_UeTemp := FALSE;
   BB1_UeSP.Stoerung.St_Leck := FALSE;
   BB1_UeSP.Stoerung.St_UeLM := FALSE;
   BB1_UeSP.Stoerung.St_UeLE := FALSE;
   BB1_UeSP.Stoerung.St_Kom_DP := FALSE;
   BB1_UeSP.Stoerung.St_Kom_int := FALSE;
   BB1_UeSP.Stoerung.St_int := FALSE;
   BB1_UeSP.Stoerung.St_LZ := FALSE;
   BB1_UeSP.Stoerung.St_BefLZ := FALSE;
   BB1_UeSP.Stoerung.Wa_EZ := FALSE;
   BB1_UeSP.Stoerung.Wa_Wart := FALSE;
   BB1_UeSP.Stoerung.St_Strm := FALSE;
   BB1_UeSP.Stoerung.Res_19 := FALSE;
   BB1_UeSP.Stoerung.Res_20 := FALSE;
   BB1_UeSP.Stoerung.Res_21 := FALSE;
   BB1_UeSP.Stoerung.Res_22 := FALSE;
   BB1_UeSP.Stoerung.Res_23 := FALSE;
   BB1_UeSP.Stoerung.Res_24 := FALSE;
   BB1_UeSP.Stoerung.Res_25 := FALSE;
   BB1_UeSP.Stoerung.Res_26 := FALSE;
   BB1_UeSP.Stoerung.Res_27 := FALSE;
   BB1_UeSP.Stoerung.Res_28 := FALSE;
   BB1_UeSP.Stoerung.Res_29 := FALSE;
   BB1_UeSP.Stoerung.Res_30 := FALSE;
   BB1_UeSP.Stoerung.Res_31 := FALSE;
   BB1_UeSP.MW_I := 0.0;
   BB1_UeSP.MW_P := 0.0;
   BB1_UeSP.EZ := 0;
   BB1_UeSP.BZ_akt := 159;
   BB1_UeSP.BZ_ges := 53465;
   BB1_UeSP.AZ_akt := 92507;
   BB1_UeSP.ESH := 122;
   BB1_UeSP.SW_akt := 0.0;
   BB1_UeSP.SW_Auto := 0.0;
   BB1_UeSP.SW_out := 0.0;
   BB1_AS1.Status.Bed_vOrt := FALSE;
   BB1_AS1.Status.Bed_UV := FALSE;
   BB1_AS1.Status.Bed_NHV := FALSE;
   BB1_AS1.Status.Bed_PLS := TRUE;
   BB1_AS1.Status.BA_Hand := FALSE;
   BB1_AS1.Status.BA_Auto := TRUE;
   BB1_AS1.Status.RB_Ein1 := FALSE;
   BB1_AS1.Status.RB_Ein2 := FALSE;
   BB1_AS1.Status.RB_Aus := TRUE;
   BB1_AS1.Status.BFR_NS := FALSE;
   BB1_AS1.Status.BFR_ECS := FALSE;
   BB1_AS1.Status.BFR_ESK := FALSE;
   BB1_AS1.Status.BFR_MAZ := FALSE;
   BB1_AS1.Status.BFR_Rev := FALSE;
   BB1_AS1.Status.BFR_Ein1 := FALSE;
   BB1_AS1.Status.BFR_Ein2 := FALSE;
   BB1_AS1.Status.BM_Ein1 := FALSE;
   BB1_AS1.Status.BM_Ein2 := FALSE;
   BB1_AS1.Status.BM_Auf := TRUE;
   BB1_AS1.Status.BM_Zu := FALSE;
   BB1_AS1.Status.BM_Ein := FALSE;
   BB1_AS1.Status.BM_Aus := TRUE;
   BB1_AS1.Status.BM_Anst1 := FALSE;
   BB1_AS1.Status.BM_Anst2 := FALSE;
   BB1_AS1.Status.BM_Auto1 := TRUE;
   BB1_AS1.Status.BM_Auto2 := FALSE;
   BB1_AS1.Status.Res_26 := FALSE;
   BB1_AS1.Status.Res_27 := FALSE;
   BB1_AS1.Status.BB_NA := FALSE;
   BB1_AS1.Status.BB_AutoOk := TRUE;
   BB1_AS1.Status.BB_SS := FALSE;
   BB1_AS1.Status.BB_SSnq := FALSE;
   BB1_AS1.Stoerung.St_allg := FALSE;
   BB1_AS1.Stoerung.St_DMA := FALSE;
   BB1_AS1.Stoerung.St_DMZ := FALSE;
   BB1_AS1.Stoerung.St_FU := FALSE;
   BB1_AS1.Stoerung.St_TL := FALSE;
   BB1_AS1.Stoerung.St_UDr := FALSE;
   BB1_AS1.Stoerung.St_UeDr := FALSE;
   BB1_AS1.Stoerung.St_UeTemp := FALSE;
   BB1_AS1.Stoerung.St_Leck := FALSE;
   BB1_AS1.Stoerung.St_UeLM := FALSE;
   BB1_AS1.Stoerung.St_UeLE := FALSE;
   BB1_AS1.Stoerung.St_Kom_DP := FALSE;
   BB1_AS1.Stoerung.St_Kom_int := FALSE;
   BB1_AS1.Stoerung.St_int := FALSE;
   BB1_AS1.Stoerung.St_LZ := FALSE;
   BB1_AS1.Stoerung.St_BefLZ := FALSE;
   BB1_AS1.Stoerung.Wa_EZ := FALSE;
   BB1_AS1.Stoerung.Wa_Wart := FALSE;
   BB1_AS1.Stoerung.St_Strm := FALSE;
   BB1_AS1.Stoerung.Res_19 := FALSE;
   BB1_AS1.Stoerung.Res_20 := FALSE;
   BB1_AS1.Stoerung.Res_21 := FALSE;
   BB1_AS1.Stoerung.Res_22 := FALSE;
   BB1_AS1.Stoerung.Res_23 := FALSE;
   BB1_AS1.Stoerung.Res_24 := FALSE;
   BB1_AS1.Stoerung.Res_25 := FALSE;
   BB1_AS1.Stoerung.Res_26 := FALSE;
   BB1_AS1.Stoerung.Res_27 := FALSE;
   BB1_AS1.Stoerung.Res_28 := FALSE;
   BB1_AS1.Stoerung.Res_29 := FALSE;
   BB1_AS1.Stoerung.Res_30 := FALSE;
   BB1_AS1.Stoerung.Res_31 := FALSE;
   BB1_AS1.MW_I := 0.0;
   BB1_AS1.MW_P := 0.0;
   BB1_AS1.EZ := 0;
   BB1_AS1.BZ_akt := 25;
   BB1_AS1.BZ_ges := 904880;
   BB1_AS1.AZ_akt := 2160;
   BB1_AS1.ESH := 35306;
   BB1_AS1.SW_akt := 0.0;
   BB1_AS1.SW_Auto := 0.0;
   BB1_AS1.SW_out := 0.0;
   BB1_AS2.Status.Bed_vOrt := FALSE;
   BB1_AS2.Status.Bed_UV := FALSE;
   BB1_AS2.Status.Bed_NHV := FALSE;
   BB1_AS2.Status.Bed_PLS := TRUE;
   BB1_AS2.Status.BA_Hand := FALSE;
   BB1_AS2.Status.BA_Auto := TRUE;
   BB1_AS2.Status.RB_Ein1 := FALSE;
   BB1_AS2.Status.RB_Ein2 := FALSE;
   BB1_AS2.Status.RB_Aus := TRUE;
   BB1_AS2.Status.BFR_NS := FALSE;
   BB1_AS2.Status.BFR_ECS := FALSE;
   BB1_AS2.Status.BFR_ESK := FALSE;
   BB1_AS2.Status.BFR_MAZ := FALSE;
   BB1_AS2.Status.BFR_Rev := FALSE;
   BB1_AS2.Status.BFR_Ein1 := FALSE;
   BB1_AS2.Status.BFR_Ein2 := FALSE;
   BB1_AS2.Status.BM_Ein1 := FALSE;
   BB1_AS2.Status.BM_Ein2 := FALSE;
   BB1_AS2.Status.BM_Auf := FALSE;
   BB1_AS2.Status.BM_Zu := TRUE;
   BB1_AS2.Status.BM_Ein := FALSE;
   BB1_AS2.Status.BM_Aus := TRUE;
   BB1_AS2.Status.BM_Anst1 := FALSE;
   BB1_AS2.Status.BM_Anst2 := FALSE;
   BB1_AS2.Status.BM_Auto1 := FALSE;
   BB1_AS2.Status.BM_Auto2 := TRUE;
   BB1_AS2.Status.Res_26 := FALSE;
   BB1_AS2.Status.Res_27 := FALSE;
   BB1_AS2.Status.BB_NA := FALSE;
   BB1_AS2.Status.BB_AutoOk := TRUE;
   BB1_AS2.Status.BB_SS := FALSE;
   BB1_AS2.Status.BB_SSnq := FALSE;
   BB1_AS2.Stoerung.St_allg := FALSE;
   BB1_AS2.Stoerung.St_DMA := FALSE;
   BB1_AS2.Stoerung.St_DMZ := FALSE;
   BB1_AS2.Stoerung.St_FU := FALSE;
   BB1_AS2.Stoerung.St_TL := FALSE;
   BB1_AS2.Stoerung.St_UDr := FALSE;
   BB1_AS2.Stoerung.St_UeDr := FALSE;
   BB1_AS2.Stoerung.St_UeTemp := FALSE;
   BB1_AS2.Stoerung.St_Leck := FALSE;
   BB1_AS2.Stoerung.St_UeLM := FALSE;
   BB1_AS2.Stoerung.St_UeLE := FALSE;
   BB1_AS2.Stoerung.St_Kom_DP := FALSE;
   BB1_AS2.Stoerung.St_Kom_int := FALSE;
   BB1_AS2.Stoerung.St_int := FALSE;
   BB1_AS2.Stoerung.St_LZ := FALSE;
   BB1_AS2.Stoerung.St_BefLZ := FALSE;
   BB1_AS2.Stoerung.Wa_EZ := FALSE;
   BB1_AS2.Stoerung.Wa_Wart := FALSE;
   BB1_AS2.Stoerung.St_Strm := FALSE;
   BB1_AS2.Stoerung.Res_19 := FALSE;
   BB1_AS2.Stoerung.Res_20 := FALSE;
   BB1_AS2.Stoerung.Res_21 := FALSE;
   BB1_AS2.Stoerung.Res_22 := FALSE;
   BB1_AS2.Stoerung.Res_23 := FALSE;
   BB1_AS2.Stoerung.Res_24 := FALSE;
   BB1_AS2.Stoerung.Res_25 := FALSE;
   BB1_AS2.Stoerung.Res_26 := FALSE;
   BB1_AS2.Stoerung.Res_27 := FALSE;
   BB1_AS2.Stoerung.Res_28 := FALSE;
   BB1_AS2.Stoerung.Res_29 := FALSE;
   BB1_AS2.Stoerung.Res_30 := FALSE;
   BB1_AS2.Stoerung.Res_31 := FALSE;
   BB1_AS2.MW_I := 0.0;
   BB1_AS2.MW_P := 0.0;
   BB1_AS2.EZ := 0;
   BB1_AS2.BZ_akt := 14;
   BB1_AS2.BZ_ges := 476867;
   BB1_AS2.AZ_akt := 2146;
   BB1_AS2.ESH := 35371;
   BB1_AS2.SW_akt := 0.0;
   BB1_AS2.SW_Auto := 0.0;
   BB1_AS2.SW_out := 0.0;
   BB1_SR1.Status.Bed_vOrt := FALSE;
   BB1_SR1.Status.Bed_UV := FALSE;
   BB1_SR1.Status.Bed_NHV := FALSE;
   BB1_SR1.Status.Bed_PLS := TRUE;
   BB1_SR1.Status.BA_Hand := FALSE;
   BB1_SR1.Status.BA_Auto := TRUE;
   BB1_SR1.Status.RB_Ein1 := FALSE;
   BB1_SR1.Status.RB_Ein2 := FALSE;
   BB1_SR1.Status.RB_Aus := TRUE;
   BB1_SR1.Status.BFR_NS := FALSE;
   BB1_SR1.Status.BFR_ECS := FALSE;
   BB1_SR1.Status.BFR_ESK := FALSE;
   BB1_SR1.Status.BFR_MAZ := FALSE;
   BB1_SR1.Status.BFR_Rev := FALSE;
   BB1_SR1.Status.BFR_Ein1 := FALSE;
   BB1_SR1.Status.BFR_Ein2 := FALSE;
   BB1_SR1.Status.BM_Ein1 := FALSE;
   BB1_SR1.Status.BM_Ein2 := FALSE;
   BB1_SR1.Status.BM_Auf := FALSE;
   BB1_SR1.Status.BM_Zu := TRUE;
   BB1_SR1.Status.BM_Ein := FALSE;
   BB1_SR1.Status.BM_Aus := TRUE;
   BB1_SR1.Status.BM_Anst1 := FALSE;
   BB1_SR1.Status.BM_Anst2 := FALSE;
   BB1_SR1.Status.BM_Auto1 := FALSE;
   BB1_SR1.Status.BM_Auto2 := TRUE;
   BB1_SR1.Status.Res_26 := FALSE;
   BB1_SR1.Status.Res_27 := FALSE;
   BB1_SR1.Status.BB_NA := FALSE;
   BB1_SR1.Status.BB_AutoOk := TRUE;
   BB1_SR1.Status.BB_SS := FALSE;
   BB1_SR1.Status.BB_SSnq := FALSE;
   BB1_SR1.Stoerung.St_allg := FALSE;
   BB1_SR1.Stoerung.St_DMA := FALSE;
   BB1_SR1.Stoerung.St_DMZ := FALSE;
   BB1_SR1.Stoerung.St_FU := FALSE;
   BB1_SR1.Stoerung.St_TL := FALSE;
   BB1_SR1.Stoerung.St_UDr := FALSE;
   BB1_SR1.Stoerung.St_UeDr := FALSE;
   BB1_SR1.Stoerung.St_UeTemp := FALSE;
   BB1_SR1.Stoerung.St_Leck := FALSE;
   BB1_SR1.Stoerung.St_UeLM := FALSE;
   BB1_SR1.Stoerung.St_UeLE := FALSE;
   BB1_SR1.Stoerung.St_Kom_DP := FALSE;
   BB1_SR1.Stoerung.St_Kom_int := FALSE;
   BB1_SR1.Stoerung.St_int := FALSE;
   BB1_SR1.Stoerung.St_LZ := FALSE;
   BB1_SR1.Stoerung.St_BefLZ := FALSE;
   BB1_SR1.Stoerung.Wa_EZ := FALSE;
   BB1_SR1.Stoerung.Wa_Wart := FALSE;
   BB1_SR1.Stoerung.St_Strm := FALSE;
   BB1_SR1.Stoerung.Res_19 := FALSE;
   BB1_SR1.Stoerung.Res_20 := FALSE;
   BB1_SR1.Stoerung.Res_21 := FALSE;
   BB1_SR1.Stoerung.Res_22 := FALSE;
   BB1_SR1.Stoerung.Res_23 := FALSE;
   BB1_SR1.Stoerung.Res_24 := FALSE;
   BB1_SR1.Stoerung.Res_25 := FALSE;
   BB1_SR1.Stoerung.Res_26 := FALSE;
   BB1_SR1.Stoerung.Res_27 := FALSE;
   BB1_SR1.Stoerung.Res_28 := FALSE;
   BB1_SR1.Stoerung.Res_29 := FALSE;
   BB1_SR1.Stoerung.Res_30 := FALSE;
   BB1_SR1.Stoerung.Res_31 := FALSE;
   BB1_SR1.MW_I := 0.0;
   BB1_SR1.MW_P := 0.0;
   BB1_SR1.EZ := 0;
   BB1_SR1.BZ_akt := 180;
   BB1_SR1.BZ_ges := 3239638;
   BB1_SR1.AZ_akt := 2005;
   BB1_SR1.ESH := 17562;
   BB1_SR1.SW_akt := 0.0;
   BB1_SR1.SW_Auto := 0.0;
   BB1_SR1.SW_out := 0.0;
   BB1_SR2.Status.Bed_vOrt := FALSE;
   BB1_SR2.Status.Bed_UV := FALSE;
   BB1_SR2.Status.Bed_NHV := FALSE;
   BB1_SR2.Status.Bed_PLS := TRUE;
   BB1_SR2.Status.BA_Hand := FALSE;
   BB1_SR2.Status.BA_Auto := TRUE;
   BB1_SR2.Status.RB_Ein1 := FALSE;
   BB1_SR2.Status.RB_Ein2 := FALSE;
   BB1_SR2.Status.RB_Aus := TRUE;
   BB1_SR2.Status.BFR_NS := FALSE;
   BB1_SR2.Status.BFR_ECS := FALSE;
   BB1_SR2.Status.BFR_ESK := FALSE;
   BB1_SR2.Status.BFR_MAZ := FALSE;
   BB1_SR2.Status.BFR_Rev := FALSE;
   BB1_SR2.Status.BFR_Ein1 := FALSE;
   BB1_SR2.Status.BFR_Ein2 := FALSE;
   BB1_SR2.Status.BM_Ein1 := FALSE;
   BB1_SR2.Status.BM_Ein2 := FALSE;
   BB1_SR2.Status.BM_Auf := FALSE;
   BB1_SR2.Status.BM_Zu := TRUE;
   BB1_SR2.Status.BM_Ein := FALSE;
   BB1_SR2.Status.BM_Aus := TRUE;
   BB1_SR2.Status.BM_Anst1 := FALSE;
   BB1_SR2.Status.BM_Anst2 := FALSE;
   BB1_SR2.Status.BM_Auto1 := FALSE;
   BB1_SR2.Status.BM_Auto2 := TRUE;
   BB1_SR2.Status.Res_26 := FALSE;
   BB1_SR2.Status.Res_27 := FALSE;
   BB1_SR2.Status.BB_NA := FALSE;
   BB1_SR2.Status.BB_AutoOk := TRUE;
   BB1_SR2.Status.BB_SS := FALSE;
   BB1_SR2.Status.BB_SSnq := FALSE;
   BB1_SR2.Stoerung.St_allg := FALSE;
   BB1_SR2.Stoerung.St_DMA := FALSE;
   BB1_SR2.Stoerung.St_DMZ := FALSE;
   BB1_SR2.Stoerung.St_FU := FALSE;
   BB1_SR2.Stoerung.St_TL := FALSE;
   BB1_SR2.Stoerung.St_UDr := FALSE;
   BB1_SR2.Stoerung.St_UeDr := FALSE;
   BB1_SR2.Stoerung.St_UeTemp := FALSE;
   BB1_SR2.Stoerung.St_Leck := FALSE;
   BB1_SR2.Stoerung.St_UeLM := FALSE;
   BB1_SR2.Stoerung.St_UeLE := FALSE;
   BB1_SR2.Stoerung.St_Kom_DP := FALSE;
   BB1_SR2.Stoerung.St_Kom_int := FALSE;
   BB1_SR2.Stoerung.St_int := FALSE;
   BB1_SR2.Stoerung.St_LZ := FALSE;
   BB1_SR2.Stoerung.St_BefLZ := FALSE;
   BB1_SR2.Stoerung.Wa_EZ := FALSE;
   BB1_SR2.Stoerung.Wa_Wart := FALSE;
   BB1_SR2.Stoerung.St_Strm := FALSE;
   BB1_SR2.Stoerung.Res_19 := FALSE;
   BB1_SR2.Stoerung.Res_20 := FALSE;
   BB1_SR2.Stoerung.Res_21 := FALSE;
   BB1_SR2.Stoerung.Res_22 := FALSE;
   BB1_SR2.Stoerung.Res_23 := FALSE;
   BB1_SR2.Stoerung.Res_24 := FALSE;
   BB1_SR2.Stoerung.Res_25 := FALSE;
   BB1_SR2.Stoerung.Res_26 := FALSE;
   BB1_SR2.Stoerung.Res_27 := FALSE;
   BB1_SR2.Stoerung.Res_28 := FALSE;
   BB1_SR2.Stoerung.Res_29 := FALSE;
   BB1_SR2.Stoerung.Res_30 := FALSE;
   BB1_SR2.Stoerung.Res_31 := FALSE;
   BB1_SR2.MW_I := 0.0;
   BB1_SR2.MW_P := 0.0;
   BB1_SR2.EZ := 0;
   BB1_SR2.BZ_akt := 181;
   BB1_SR2.BZ_ges := 3160108;
   BB1_SR2.AZ_akt := 5605;
   BB1_SR2.ESH := 17582;
   BB1_SR2.SW_akt := 0.0;
   BB1_SR2.SW_Auto := 0.0;
   BB1_SR2.SW_out := 0.0;
   BB2_RZP1.Status.Bed_vOrt := FALSE;
   BB2_RZP1.Status.Bed_UV := FALSE;
   BB2_RZP1.Status.Bed_NHV := FALSE;
   BB2_RZP1.Status.Bed_PLS := TRUE;
   BB2_RZP1.Status.BA_Hand := FALSE;
   BB2_RZP1.Status.BA_Auto := TRUE;
   BB2_RZP1.Status.RB_Ein1 := FALSE;
   BB2_RZP1.Status.RB_Ein2 := FALSE;
   BB2_RZP1.Status.RB_Aus := TRUE;
   BB2_RZP1.Status.BFR_NS := FALSE;
   BB2_RZP1.Status.BFR_ECS := FALSE;
   BB2_RZP1.Status.BFR_ESK := FALSE;
   BB2_RZP1.Status.BFR_MAZ := FALSE;
   BB2_RZP1.Status.BFR_Rev := FALSE;
   BB2_RZP1.Status.BFR_Ein1 := FALSE;
   BB2_RZP1.Status.BFR_Ein2 := FALSE;
   BB2_RZP1.Status.BM_Ein1 := FALSE;
   BB2_RZP1.Status.BM_Ein2 := FALSE;
   BB2_RZP1.Status.BM_Auf := FALSE;
   BB2_RZP1.Status.BM_Zu := FALSE;
   BB2_RZP1.Status.BM_Ein := FALSE;
   BB2_RZP1.Status.BM_Aus := TRUE;
   BB2_RZP1.Status.BM_Anst1 := FALSE;
   BB2_RZP1.Status.BM_Anst2 := FALSE;
   BB2_RZP1.Status.BM_Auto1 := FALSE;
   BB2_RZP1.Status.BM_Auto2 := FALSE;
   BB2_RZP1.Status.Res_26 := FALSE;
   BB2_RZP1.Status.Res_27 := FALSE;
   BB2_RZP1.Status.BB_NA := FALSE;
   BB2_RZP1.Status.BB_AutoOk := TRUE;
   BB2_RZP1.Status.BB_SS := FALSE;
   BB2_RZP1.Status.BB_SSnq := FALSE;
   BB2_RZP1.Stoerung.St_allg := FALSE;
   BB2_RZP1.Stoerung.St_DMA := FALSE;
   BB2_RZP1.Stoerung.St_DMZ := FALSE;
   BB2_RZP1.Stoerung.St_FU := FALSE;
   BB2_RZP1.Stoerung.St_TL := FALSE;
   BB2_RZP1.Stoerung.St_UDr := FALSE;
   BB2_RZP1.Stoerung.St_UeDr := FALSE;
   BB2_RZP1.Stoerung.St_UeTemp := FALSE;
   BB2_RZP1.Stoerung.St_Leck := FALSE;
   BB2_RZP1.Stoerung.St_UeLM := FALSE;
   BB2_RZP1.Stoerung.St_UeLE := FALSE;
   BB2_RZP1.Stoerung.St_Kom_DP := FALSE;
   BB2_RZP1.Stoerung.St_Kom_int := FALSE;
   BB2_RZP1.Stoerung.St_int := FALSE;
   BB2_RZP1.Stoerung.St_LZ := FALSE;
   BB2_RZP1.Stoerung.St_BefLZ := FALSE;
   BB2_RZP1.Stoerung.Wa_EZ := FALSE;
   BB2_RZP1.Stoerung.Wa_Wart := FALSE;
   BB2_RZP1.Stoerung.St_Strm := FALSE;
   BB2_RZP1.Stoerung.Res_19 := FALSE;
   BB2_RZP1.Stoerung.Res_20 := FALSE;
   BB2_RZP1.Stoerung.Res_21 := FALSE;
   BB2_RZP1.Stoerung.Res_22 := FALSE;
   BB2_RZP1.Stoerung.Res_23 := FALSE;
   BB2_RZP1.Stoerung.Res_24 := FALSE;
   BB2_RZP1.Stoerung.Res_25 := FALSE;
   BB2_RZP1.Stoerung.Res_26 := FALSE;
   BB2_RZP1.Stoerung.Res_27 := FALSE;
   BB2_RZP1.Stoerung.Res_28 := FALSE;
   BB2_RZP1.Stoerung.Res_29 := FALSE;
   BB2_RZP1.Stoerung.Res_30 := FALSE;
   BB2_RZP1.Stoerung.Res_31 := FALSE;
   BB2_RZP1.MW_I := 0.0;
   BB2_RZP1.MW_P := 0.0;
   BB2_RZP1.EZ := 0;
   BB2_RZP1.BZ_akt := 844;
   BB2_RZP1.BZ_ges := 114029;
   BB2_RZP1.AZ_akt := 1265;
   BB2_RZP1.ESH := 135;
   BB2_RZP1.SW_akt := 0.0;
   BB2_RZP1.SW_Auto := 0.0;
   BB2_RZP1.SW_out := 0.0;
   BB2_RZP2.Status.Bed_vOrt := FALSE;
   BB2_RZP2.Status.Bed_UV := FALSE;
   BB2_RZP2.Status.Bed_NHV := FALSE;
   BB2_RZP2.Status.Bed_PLS := TRUE;
   BB2_RZP2.Status.BA_Hand := FALSE;
   BB2_RZP2.Status.BA_Auto := TRUE;
   BB2_RZP2.Status.RB_Ein1 := FALSE;
   BB2_RZP2.Status.RB_Ein2 := FALSE;
   BB2_RZP2.Status.RB_Aus := TRUE;
   BB2_RZP2.Status.BFR_NS := FALSE;
   BB2_RZP2.Status.BFR_ECS := FALSE;
   BB2_RZP2.Status.BFR_ESK := FALSE;
   BB2_RZP2.Status.BFR_MAZ := FALSE;
   BB2_RZP2.Status.BFR_Rev := FALSE;
   BB2_RZP2.Status.BFR_Ein1 := FALSE;
   BB2_RZP2.Status.BFR_Ein2 := FALSE;
   BB2_RZP2.Status.BM_Ein1 := FALSE;
   BB2_RZP2.Status.BM_Ein2 := FALSE;
   BB2_RZP2.Status.BM_Auf := FALSE;
   BB2_RZP2.Status.BM_Zu := FALSE;
   BB2_RZP2.Status.BM_Ein := FALSE;
   BB2_RZP2.Status.BM_Aus := TRUE;
   BB2_RZP2.Status.BM_Anst1 := FALSE;
   BB2_RZP2.Status.BM_Anst2 := FALSE;
   BB2_RZP2.Status.BM_Auto1 := FALSE;
   BB2_RZP2.Status.BM_Auto2 := FALSE;
   BB2_RZP2.Status.Res_26 := FALSE;
   BB2_RZP2.Status.Res_27 := FALSE;
   BB2_RZP2.Status.BB_NA := FALSE;
   BB2_RZP2.Status.BB_AutoOk := TRUE;
   BB2_RZP2.Status.BB_SS := FALSE;
   BB2_RZP2.Status.BB_SSnq := FALSE;
   BB2_RZP2.Stoerung.St_allg := FALSE;
   BB2_RZP2.Stoerung.St_DMA := FALSE;
   BB2_RZP2.Stoerung.St_DMZ := FALSE;
   BB2_RZP2.Stoerung.St_FU := FALSE;
   BB2_RZP2.Stoerung.St_TL := FALSE;
   BB2_RZP2.Stoerung.St_UDr := FALSE;
   BB2_RZP2.Stoerung.St_UeDr := FALSE;
   BB2_RZP2.Stoerung.St_UeTemp := FALSE;
   BB2_RZP2.Stoerung.St_Leck := FALSE;
   BB2_RZP2.Stoerung.St_UeLM := FALSE;
   BB2_RZP2.Stoerung.St_UeLE := FALSE;
   BB2_RZP2.Stoerung.St_Kom_DP := FALSE;
   BB2_RZP2.Stoerung.St_Kom_int := FALSE;
   BB2_RZP2.Stoerung.St_int := FALSE;
   BB2_RZP2.Stoerung.St_LZ := FALSE;
   BB2_RZP2.Stoerung.St_BefLZ := FALSE;
   BB2_RZP2.Stoerung.Wa_EZ := FALSE;
   BB2_RZP2.Stoerung.Wa_Wart := FALSE;
   BB2_RZP2.Stoerung.St_Strm := FALSE;
   BB2_RZP2.Stoerung.Res_19 := FALSE;
   BB2_RZP2.Stoerung.Res_20 := FALSE;
   BB2_RZP2.Stoerung.Res_21 := FALSE;
   BB2_RZP2.Stoerung.Res_22 := FALSE;
   BB2_RZP2.Stoerung.Res_23 := FALSE;
   BB2_RZP2.Stoerung.Res_24 := FALSE;
   BB2_RZP2.Stoerung.Res_25 := FALSE;
   BB2_RZP2.Stoerung.Res_26 := FALSE;
   BB2_RZP2.Stoerung.Res_27 := FALSE;
   BB2_RZP2.Stoerung.Res_28 := FALSE;
   BB2_RZP2.Stoerung.Res_29 := FALSE;
   BB2_RZP2.Stoerung.Res_30 := FALSE;
   BB2_RZP2.Stoerung.Res_31 := FALSE;
   BB2_RZP2.MW_I := 0.0;
   BB2_RZP2.MW_P := 0.0;
   BB2_RZP2.EZ := 0;
   BB2_RZP2.BZ_akt := 845;
   BB2_RZP2.BZ_ges := 113176;
   BB2_RZP2.AZ_akt := 4864;
   BB2_RZP2.ESH := 134;
   BB2_RZP2.SW_akt := 0.0;
   BB2_RZP2.SW_Auto := 0.0;
   BB2_RZP2.SW_out := 0.0;
   BB2_UeSP.Status.Bed_vOrt := FALSE;
   BB2_UeSP.Status.Bed_UV := FALSE;
   BB2_UeSP.Status.Bed_NHV := FALSE;
   BB2_UeSP.Status.Bed_PLS := TRUE;
   BB2_UeSP.Status.BA_Hand := FALSE;
   BB2_UeSP.Status.BA_Auto := TRUE;
   BB2_UeSP.Status.RB_Ein1 := FALSE;
   BB2_UeSP.Status.RB_Ein2 := FALSE;
   BB2_UeSP.Status.RB_Aus := TRUE;
   BB2_UeSP.Status.BFR_NS := FALSE;
   BB2_UeSP.Status.BFR_ECS := FALSE;
   BB2_UeSP.Status.BFR_ESK := FALSE;
   BB2_UeSP.Status.BFR_MAZ := FALSE;
   BB2_UeSP.Status.BFR_Rev := FALSE;
   BB2_UeSP.Status.BFR_Ein1 := FALSE;
   BB2_UeSP.Status.BFR_Ein2 := FALSE;
   BB2_UeSP.Status.BM_Ein1 := FALSE;
   BB2_UeSP.Status.BM_Ein2 := FALSE;
   BB2_UeSP.Status.BM_Auf := FALSE;
   BB2_UeSP.Status.BM_Zu := FALSE;
   BB2_UeSP.Status.BM_Ein := FALSE;
   BB2_UeSP.Status.BM_Aus := TRUE;
   BB2_UeSP.Status.BM_Anst1 := FALSE;
   BB2_UeSP.Status.BM_Anst2 := FALSE;
   BB2_UeSP.Status.BM_Auto1 := FALSE;
   BB2_UeSP.Status.BM_Auto2 := FALSE;
   BB2_UeSP.Status.Res_26 := FALSE;
   BB2_UeSP.Status.Res_27 := FALSE;
   BB2_UeSP.Status.BB_NA := FALSE;
   BB2_UeSP.Status.BB_AutoOk := TRUE;
   BB2_UeSP.Status.BB_SS := FALSE;
   BB2_UeSP.Status.BB_SSnq := FALSE;
   BB2_UeSP.Stoerung.St_allg := FALSE;
   BB2_UeSP.Stoerung.St_DMA := FALSE;
   BB2_UeSP.Stoerung.St_DMZ := FALSE;
   BB2_UeSP.Stoerung.St_FU := FALSE;
   BB2_UeSP.Stoerung.St_TL := FALSE;
   BB2_UeSP.Stoerung.St_UDr := FALSE;
   BB2_UeSP.Stoerung.St_UeDr := FALSE;
   BB2_UeSP.Stoerung.St_UeTemp := FALSE;
   BB2_UeSP.Stoerung.St_Leck := FALSE;
   BB2_UeSP.Stoerung.St_UeLM := FALSE;
   BB2_UeSP.Stoerung.St_UeLE := FALSE;
   BB2_UeSP.Stoerung.St_Kom_DP := FALSE;
   BB2_UeSP.Stoerung.St_Kom_int := FALSE;
   BB2_UeSP.Stoerung.St_int := FALSE;
   BB2_UeSP.Stoerung.St_LZ := FALSE;
   BB2_UeSP.Stoerung.St_BefLZ := FALSE;
   BB2_UeSP.Stoerung.Wa_EZ := FALSE;
   BB2_UeSP.Stoerung.Wa_Wart := FALSE;
   BB2_UeSP.Stoerung.St_Strm := FALSE;
   BB2_UeSP.Stoerung.Res_19 := FALSE;
   BB2_UeSP.Stoerung.Res_20 := FALSE;
   BB2_UeSP.Stoerung.Res_21 := FALSE;
   BB2_UeSP.Stoerung.Res_22 := FALSE;
   BB2_UeSP.Stoerung.Res_23 := FALSE;
   BB2_UeSP.Stoerung.Res_24 := FALSE;
   BB2_UeSP.Stoerung.Res_25 := FALSE;
   BB2_UeSP.Stoerung.Res_26 := FALSE;
   BB2_UeSP.Stoerung.Res_27 := FALSE;
   BB2_UeSP.Stoerung.Res_28 := FALSE;
   BB2_UeSP.Stoerung.Res_29 := FALSE;
   BB2_UeSP.Stoerung.Res_30 := FALSE;
   BB2_UeSP.Stoerung.Res_31 := FALSE;
   BB2_UeSP.MW_I := 0.0;
   BB2_UeSP.MW_P := 0.0;
   BB2_UeSP.EZ := 0;
   BB2_UeSP.BZ_akt := 288;
   BB2_UeSP.BZ_ges := 35887;
   BB2_UeSP.AZ_akt := 95956;
   BB2_UeSP.ESH := 122;
   BB2_UeSP.SW_akt := 0.0;
   BB2_UeSP.SW_Auto := 0.0;
   BB2_UeSP.SW_out := 0.0;
   BB2_AS1.Status.Bed_vOrt := FALSE;
   BB2_AS1.Status.Bed_UV := FALSE;
   BB2_AS1.Status.Bed_NHV := FALSE;
   BB2_AS1.Status.Bed_PLS := TRUE;
   BB2_AS1.Status.BA_Hand := FALSE;
   BB2_AS1.Status.BA_Auto := TRUE;
   BB2_AS1.Status.RB_Ein1 := FALSE;
   BB2_AS1.Status.RB_Ein2 := FALSE;
   BB2_AS1.Status.RB_Aus := TRUE;
   BB2_AS1.Status.BFR_NS := FALSE;
   BB2_AS1.Status.BFR_ECS := FALSE;
   BB2_AS1.Status.BFR_ESK := FALSE;
   BB2_AS1.Status.BFR_MAZ := FALSE;
   BB2_AS1.Status.BFR_Rev := FALSE;
   BB2_AS1.Status.BFR_Ein1 := FALSE;
   BB2_AS1.Status.BFR_Ein2 := FALSE;
   BB2_AS1.Status.BM_Ein1 := FALSE;
   BB2_AS1.Status.BM_Ein2 := FALSE;
   BB2_AS1.Status.BM_Auf := FALSE;
   BB2_AS1.Status.BM_Zu := TRUE;
   BB2_AS1.Status.BM_Ein := FALSE;
   BB2_AS1.Status.BM_Aus := TRUE;
   BB2_AS1.Status.BM_Anst1 := FALSE;
   BB2_AS1.Status.BM_Anst2 := FALSE;
   BB2_AS1.Status.BM_Auto1 := FALSE;
   BB2_AS1.Status.BM_Auto2 := TRUE;
   BB2_AS1.Status.Res_26 := FALSE;
   BB2_AS1.Status.Res_27 := FALSE;
   BB2_AS1.Status.BB_NA := FALSE;
   BB2_AS1.Status.BB_AutoOk := TRUE;
   BB2_AS1.Status.BB_SS := FALSE;
   BB2_AS1.Status.BB_SSnq := FALSE;
   BB2_AS1.Stoerung.St_allg := FALSE;
   BB2_AS1.Stoerung.St_DMA := FALSE;
   BB2_AS1.Stoerung.St_DMZ := FALSE;
   BB2_AS1.Stoerung.St_FU := FALSE;
   BB2_AS1.Stoerung.St_TL := FALSE;
   BB2_AS1.Stoerung.St_UDr := FALSE;
   BB2_AS1.Stoerung.St_UeDr := FALSE;
   BB2_AS1.Stoerung.St_UeTemp := FALSE;
   BB2_AS1.Stoerung.St_Leck := FALSE;
   BB2_AS1.Stoerung.St_UeLM := FALSE;
   BB2_AS1.Stoerung.St_UeLE := FALSE;
   BB2_AS1.Stoerung.St_Kom_DP := FALSE;
   BB2_AS1.Stoerung.St_Kom_int := FALSE;
   BB2_AS1.Stoerung.St_int := FALSE;
   BB2_AS1.Stoerung.St_LZ := FALSE;
   BB2_AS1.Stoerung.St_BefLZ := FALSE;
   BB2_AS1.Stoerung.Wa_EZ := FALSE;
   BB2_AS1.Stoerung.Wa_Wart := FALSE;
   BB2_AS1.Stoerung.St_Strm := FALSE;
   BB2_AS1.Stoerung.Res_19 := FALSE;
   BB2_AS1.Stoerung.Res_20 := FALSE;
   BB2_AS1.Stoerung.Res_21 := FALSE;
   BB2_AS1.Stoerung.Res_22 := FALSE;
   BB2_AS1.Stoerung.Res_23 := FALSE;
   BB2_AS1.Stoerung.Res_24 := FALSE;
   BB2_AS1.Stoerung.Res_25 := FALSE;
   BB2_AS1.Stoerung.Res_26 := FALSE;
   BB2_AS1.Stoerung.Res_27 := FALSE;
   BB2_AS1.Stoerung.Res_28 := FALSE;
   BB2_AS1.Stoerung.Res_29 := FALSE;
   BB2_AS1.Stoerung.Res_30 := FALSE;
   BB2_AS1.Stoerung.Res_31 := FALSE;
   BB2_AS1.MW_I := 0.0;
   BB2_AS1.MW_P := 0.0;
   BB2_AS1.EZ := 0;
   BB2_AS1.BZ_akt := 28;
   BB2_AS1.BZ_ges := 978804;
   BB2_AS1.AZ_akt := 2109;
   BB2_AS1.ESH := 35307;
   BB2_AS1.SW_akt := 0.0;
   BB2_AS1.SW_Auto := 0.0;
   BB2_AS1.SW_out := 0.0;
   BB2_AS2.Status.Bed_vOrt := FALSE;
   BB2_AS2.Status.Bed_UV := FALSE;
   BB2_AS2.Status.Bed_NHV := FALSE;
   BB2_AS2.Status.Bed_PLS := TRUE;
   BB2_AS2.Status.BA_Hand := FALSE;
   BB2_AS2.Status.BA_Auto := TRUE;
   BB2_AS2.Status.RB_Ein1 := FALSE;
   BB2_AS2.Status.RB_Ein2 := FALSE;
   BB2_AS2.Status.RB_Aus := TRUE;
   BB2_AS2.Status.BFR_NS := FALSE;
   BB2_AS2.Status.BFR_ECS := FALSE;
   BB2_AS2.Status.BFR_ESK := FALSE;
   BB2_AS2.Status.BFR_MAZ := FALSE;
   BB2_AS2.Status.BFR_Rev := FALSE;
   BB2_AS2.Status.BFR_Ein1 := FALSE;
   BB2_AS2.Status.BFR_Ein2 := FALSE;
   BB2_AS2.Status.BM_Ein1 := FALSE;
   BB2_AS2.Status.BM_Ein2 := FALSE;
   BB2_AS2.Status.BM_Auf := TRUE;
   BB2_AS2.Status.BM_Zu := FALSE;
   BB2_AS2.Status.BM_Ein := FALSE;
   BB2_AS2.Status.BM_Aus := TRUE;
   BB2_AS2.Status.BM_Anst1 := FALSE;
   BB2_AS2.Status.BM_Anst2 := FALSE;
   BB2_AS2.Status.BM_Auto1 := TRUE;
   BB2_AS2.Status.BM_Auto2 := FALSE;
   BB2_AS2.Status.Res_26 := FALSE;
   BB2_AS2.Status.Res_27 := FALSE;
   BB2_AS2.Status.BB_NA := FALSE;
   BB2_AS2.Status.BB_AutoOk := TRUE;
   BB2_AS2.Status.BB_SS := FALSE;
   BB2_AS2.Status.BB_SSnq := FALSE;
   BB2_AS2.Stoerung.St_allg := FALSE;
   BB2_AS2.Stoerung.St_DMA := FALSE;
   BB2_AS2.Stoerung.St_DMZ := FALSE;
   BB2_AS2.Stoerung.St_FU := FALSE;
   BB2_AS2.Stoerung.St_TL := FALSE;
   BB2_AS2.Stoerung.St_UDr := FALSE;
   BB2_AS2.Stoerung.St_UeDr := FALSE;
   BB2_AS2.Stoerung.St_UeTemp := FALSE;
   BB2_AS2.Stoerung.St_Leck := FALSE;
   BB2_AS2.Stoerung.St_UeLM := FALSE;
   BB2_AS2.Stoerung.St_UeLE := FALSE;
   BB2_AS2.Stoerung.St_Kom_DP := FALSE;
   BB2_AS2.Stoerung.St_Kom_int := FALSE;
   BB2_AS2.Stoerung.St_int := FALSE;
   BB2_AS2.Stoerung.St_LZ := FALSE;
   BB2_AS2.Stoerung.St_BefLZ := FALSE;
   BB2_AS2.Stoerung.Wa_EZ := FALSE;
   BB2_AS2.Stoerung.Wa_Wart := FALSE;
   BB2_AS2.Stoerung.St_Strm := FALSE;
   BB2_AS2.Stoerung.Res_19 := FALSE;
   BB2_AS2.Stoerung.Res_20 := FALSE;
   BB2_AS2.Stoerung.Res_21 := FALSE;
   BB2_AS2.Stoerung.Res_22 := FALSE;
   BB2_AS2.Stoerung.Res_23 := FALSE;
